LIN {X 0,Y 474.588,Z 296.363,A -85,B 0,C 180,E1 -7327.385,E2 -7327.385} C_VEL
LIN {X 0,Y 474.608,Z 296.362,A -85,B 0,C 180,E1 -7329.644,E2 -7329.644} C_VEL
LIN {X 0,Y 474.585,Z 296.364,A -85,B 0,C 180,E1 -7332.938,E2 -7332.938} C_VEL
LIN {X 0,Y 474.607,Z 296.362,A -85,B 0,C 180,E1 -7335.895,E2 -7335.895} C_VEL
LIN {X 0,Y 474.626,Z 296.36,A -85,B 0,C 180,E1 -7339.042,E2 -7339.042} C_VEL
LIN {X 0,Y 474.611,Z 296.36,A -85,B 0,C 180,E1 -7341.705,E2 -7341.705} C_VEL
LIN {X 0,Y 474.626,Z 296.367,A -85,B 0,C 180,E1 -7344.725,E2 -7344.725} C_VEL
LIN {X 0,Y 474.639,Z 296.356,A -85,B 0,C 180,E1 -7347.788,E2 -7347.788} C_VEL
LIN {X 0,Y 474.611,Z 296.367,A -85,B 0,C 180,E1 -7350.888,E2 -7350.888} C_VEL
LIN {X 0,Y 474.616,Z 296.361,A -85,B 0,C 180,E1 -7353.626,E2 -7353.626} C_VEL
LIN {X 0,Y 474.638,Z 296.358,A -85,B 0,C 180,E1 -7356.642,E2 -7356.642} C_VEL
LIN {X 0,Y 474.658,Z 296.354,A -85,B 0,C 180,E1 -7360.089,E2 -7360.089} C_VEL
LIN {X 0,Y 474.642,Z 296.357,A -85,B 0,C 180,E1 -7362.774,E2 -7362.774} C_VEL
LIN {X 0,Y 474.65,Z 296.362,A -85,B 0,C 180,E1 -7365.421,E2 -7365.421} C_VEL
LIN {X 0,Y 474.708,Z 296.351,A -85,B 0,C 180,E1 -7368.037,E2 -7368.037} C_VEL
LIN {X 0,Y 474.707,Z 296.352,A -85,B 0,C 180,E1 -7371.486,E2 -7371.486} C_VEL
LIN {X 0,Y 474.768,Z 296.347,A -85,B 0,C 180,E1 -7374.052,E2 -7374.052} C_VEL
LIN {X 0,Y 474.886,Z 296.327,A -85,B 0,C 180,E1 -7377.455,E2 -7377.455} C_VEL
LIN {X 0,Y 474.913,Z 296.33,A -85,B 0,C 180,E1 -7380,E2 -7380} C_VEL
LIN {X 0,Y 474.887,Z 296.329,A -85,B 0,C 180,E1 -7382.544,E2 -7382.544} C_VEL
LIN {X 0,Y 474.752,Z 296.346,A -85,B 0,C 180,E1 -7385.948,E2 -7385.948} C_VEL
LIN {X 0,Y 474.715,Z 296.355,A -85,B 0,C 180,E1 -7388.514,E2 -7388.514} C_VEL
LIN {X 0,Y 474.707,Z 296.349,A -85,B 0,C 180,E1 -7391.962,E2 -7391.962} C_VEL
LIN {X 0,Y 474.703,Z 296.349,A -85,B 0,C 180,E1 -7395.455,E2 -7395.455} C_VEL
LIN {X 0,Y 474.665,Z 296.359,A -85,B 0,C 180,E1 -7399.01,E2 -7399.01} C_VEL
LIN {X 0,Y 474.591,Z 296.363,A -85,B 0,C 180,E1 -7401.729,E2 -7401.729} C_VEL
LIN {X 0,Y 474.638,Z 296.358,A -85,B 0,C 180,E1 -7404.494,E2 -7404.494} C_VEL
LIN {X 0,Y 474.639,Z 296.363,A -85,B 0,C 180,E1 -7407.324,E2 -7407.324} C_VEL
LIN {X 0,Y 474.604,Z 296.361,A -85,B 0,C 180,E1 -7410.23,E2 -7410.23} C_VEL
LIN {X 0,Y 474.627,Z 296.364,A -85,B 0,C 180,E1 -7413.221,E2 -7413.221} C_VEL
LIN {X 0,Y 474.586,Z 296.363,A -85,B 0,C 180,E1 -7416.324,E2 -7416.324} C_VEL
LIN {X 0,Y 474.628,Z 296.366,A -85,B 0,C 180,E1 -7419.547,E2 -7419.547} C_VEL
LIN {X 0,Y 474.602,Z 296.363,A -85,B 0,C 180,E1 -7422.233,E2 -7422.233} C_VEL
LIN {X 0,Y 474.618,Z 296.361,A -85,B 0,C 180,E1 -7425.297,E2 -7425.297} C_VEL
LIN {X 0,Y 474.616,Z 296.364,A -85,B 0,C 180,E1 -7428.214,E2 -7428.214} C_VEL
LIN {X 0,Y 474.61,Z 296.362,A -85,B 0,C 180,E1 -7431.542,E2 -7431.542} C_VEL
LIN {X 0,Y 474.624,Z 296.36,A -85,B 0,C 180,E1 -7434.725,E2 -7434.725} C_VEL
LIN {X 0,Y 474.637,Z 296.358,A -85,B 0,C 180,E1 -7437.787,E2 -7437.787} C_VEL
LIN {X 0,Y 474.609,Z 296.363,A -85,B 0,C 180,E1 -7440.888,E2 -7440.888} C_VEL
LIN {X 0,Y 474.614,Z 296.359,A -85,B 0,C 180,E1 -7443.625,E2 -7443.625} C_VEL
LIN {X 0,Y 474.635,Z 296.366,A -85,B 0,C 180,E1 -7446.641,E2 -7446.641} C_VEL
LIN {X 0,Y 474.654,Z 296.355,A -85,B 0,C 180,E1 -7450.089,E2 -7450.089} C_VEL
LIN {X 0,Y 474.646,Z 296.356,A -85,B 0,C 180,E1 -7451.662,E2 -7451.662} C_VEL
LIN {X 0,Y 473.977,Z 296.442,A -85,B 0,C 180,E1 -7452.371,E2 -7452.371} C_VEL
LIN {X 0,Y 471.13,Z 296.799,A -85,B 0,C 180,E1 -7453.523,E2 -7453.523} C_VEL
LIN {X 0,Y 468.721,Z 297.102,A -85,B 0,C 180,E1 -7454.451,E2 -7454.451} C_VEL
LIN {X 0,Y 467.682,Z 297.229,A -85,B 0,C 180,E1 -7455.168,E2 -7455.168} C_VEL
LIN {X 0,Y 467.595,Z 297.237,A -85,B 0,C 180,E1 -7455.411,E2 -7455.411} C_VEL
LIN {X 0,Y 467.649,Z 297.23,A -85,B 0,C 180,E1 -7458.733,E2 -7458.733} C_VEL
LIN {X 0,Y 467.668,Z 297.234,A -85,B 0,C 180,E1 -7461.356,E2 -7461.356} C_VEL
LIN {X 0,Y 467.716,Z 297.278,A -85,B 0,C 180,E1 -7462.459,E2 -7462.459} C_VEL
LIN {X 0,Y 468.745,Z 303.411,A -85,B 0,C 180,E1 -7463.759,E2 -7463.759} C_VEL
LIN {X 0,Y 468.493,Z 316.288,A -85,B 0,C 180,E1 -7466.344,E2 -7466.344} C_VEL
LIN {X 0,Y 468.341,Z 320.083,A -85,B 0,C 180,E1 -7467.096,E2 -7467.096} C_VEL
LIN {X 0,Y 471.245,Z 335.027,A -85,B 0,C 180,E1 -7467.435,E2 -7467.435} C_VEL
LIN {X 0,Y 470.498,Z 427.693,A -85,B 0,C 180,E1 -7468.876,E2 -7468.876} C_VEL
LIN {X 0,Y 470.219,Z 440.684,A -85,B 0,C 180,E1 -7469.25,E2 -7469.25} C_VEL
LIN {X 0,Y 469.872,Z 453.221,A -85,B 0,C 180,E1 -7469.785,E2 -7469.785} C_VEL
LIN {X 0,Y 469.47,Z 464.404,A -85,B 0,C 180,E1 -7470.428,E2 -7470.428} C_VEL
LIN {X 0,Y 468.93,Z 475.979,A -85,B 0,C 180,E1 -7471.287,E2 -7471.287} C_VEL
LIN {X 0,Y 468.444,Z 486.385,A -85,B 0,C 180,E1 -7472.256,E2 -7472.256} C_VEL
LIN {X 0,Y 467.978,Z 494.922,A -85,B 0,C 180,E1 -7473.228,E2 -7473.228} C_VEL
LIN {X 0,Y 467.634,Z 502.784,A -85,B 0,C 180,E1 -7474.309,E2 -7474.309} C_VEL
LIN {X 0,Y 467.239,Z 510.504,A -85,B 0,C 180,E1 -7475.61,E2 -7475.61} C_VEL
LIN {X 0,Y 467.086,Z 516.68,A -85,B 0,C 180,E1 -7476.913,E2 -7476.913} C_VEL
LIN {X 0,Y 466.88,Z 521.614,A -85,B 0,C 180,E1 -7478.221,E2 -7478.221} C_VEL
LIN {X 0,Y 466.723,Z 525.428,A -85,B 0,C 180,E1 -7479.534,E2 -7479.534} C_VEL
LIN {X 0,Y 466.689,Z 527.392,A -85,B 0,C 180,E1 -7480.41,E2 -7480.41} C_VEL
LIN {X 0,Y 466.645,Z 529.579,A -85,B 0,C 180,E1 -7481.779,E2 -7481.779} C_VEL
LIN {X 0,Y 466.555,Z 530.699,A -85,B 0,C 180,E1 -7483.058,E2 -7483.058} C_VEL
LIN {X 0,Y 466.525,Z 530.982,A -85,B 0,C 180,E1 -7483.947,E2 -7483.947} C_VEL
LIN {X 0,Y 466.613,Z 530.508,A -85,B 0,C 180,E1 -7485.432,E2 -7485.432} C_VEL
LIN {X 0,Y 466.545,Z 529.246,A -85,B 0,C 180,E1 -7486.631,E2 -7486.631} C_VEL
LIN {X 0,Y 466.636,Z 527.819,A -85,B 0,C 180,E1 -7487.53,E2 -7487.53} C_VEL
LIN {X 0,Y 466.785,Z 524.885,A -85,B 0,C 180,E1 -7488.841,E2 -7488.841} C_VEL
LIN {X 0,Y 466.937,Z 520.549,A -85,B 0,C 180,E1 -7490.253,E2 -7490.253} C_VEL
LIN {X 0,Y 467.135,Z 515.016,A -85,B 0,C 180,E1 -7491.628,E2 -7491.628} C_VEL
LIN {X 0,Y 467.489,Z 507.978,A -85,B 0,C 180,E1 -7493.008,E2 -7493.008} C_VEL
LIN {X 0,Y 467.83,Z 500.694,A -85,B 0,C 180,E1 -7494.164,E2 -7494.164} C_VEL
LIN {X 0,Y 468.293,Z 491.797,A -85,B 0,C 180,E1 -7495.322,E2 -7495.322} C_VEL
LIN {X 0,Y 468.754,Z 482.224,A -85,B 0,C 180,E1 -7496.333,E2 -7496.333} C_VEL
LIN {X 0,Y 469.341,Z 470.875,A -85,B 0,C 180,E1 -7497.295,E2 -7497.295} C_VEL
LIN {X 0,Y 469.835,Z 459.618,A -85,B 0,C 180,E1 -7498.049,E2 -7498.049} C_VEL
LIN {X 0,Y 470.194,Z 448.276,A -85,B 0,C 180,E1 -7498.635,E2 -7498.635} C_VEL
LIN {X 0,Y 470.537,Z 434.709,A -85,B 0,C 180,E1 -7499.131,E2 -7499.131} C_VEL
LIN {X 0,Y 470.768,Z 421.895,A -85,B 0,C 180,E1 -7499.422,E2 -7499.422} C_VEL
LIN {X 0,Y 471.51,Z 335.217,A -85,B 0,C 180,E1 -7500.76,E2 -7500.76} C_VEL
LIN {X 0,Y 468.488,Z 319.878,A -85,B 0,C 180,E1 -7501.148,E2 -7501.148} C_VEL
LIN {X 0,Y 468.923,Z 305.629,A -85,B 0,C 180,E1 -7503.915,E2 -7503.915} C_VEL
LIN {X 0,Y 468.16,Z 300.097,A -85,B 0,C 180,E1 -7505.043,E2 -7505.043} C_VEL
LIN {X 0,Y 467.563,Z 297.245,A -85,B 0,C 180,E1 -7505.664,E2 -7505.664} C_VEL
LIN {X 0,Y 467.546,Z 297.246,A -85,B 0,C 180,E1 -7509.147,E2 -7509.147} C_VEL
LIN {X 0,Y 467.56,Z 297.242,A -85,B 0,C 180,E1 -7511.403,E2 -7511.403} C_VEL
LIN {X 0,Y 467.558,Z 297.247,A -85,B 0,C 180,E1 -7514.947,E2 -7514.947} C_VEL
LIN {X 0,Y 467.535,Z 297.244,A -85,B 0,C 180,E1 -7517.438,E2 -7517.438} C_VEL
LIN {X 0,Y 467.555,Z 297.241,A -85,B 0,C 180,E1 -7520.048,E2 -7520.048} C_VEL
LIN {X 0,Y 467.52,Z 297.248,A -85,B 0,C 180,E1 -7523.037,E2 -7523.037} C_VEL
LIN {X 0,Y 467.558,Z 297.23,A -85,B 0,C 180,E1 -7526.21,E2 -7526.21} C_VEL
LIN {X 0,Y 467.559,Z 297.245,A -85,B 0,C 180,E1 -7529.266,E2 -7529.266} C_VEL
LIN {X 0,Y 467.594,Z 297.236,A -85,B 0,C 180,E1 -7532.469,E2 -7532.469} C_VEL
LIN {X 0,Y 467.545,Z 297.241,A -85,B 0,C 180,E1 -7535.11,E2 -7535.11} C_VEL
LIN {X 0,Y 467.524,Z 297.247,A -85,B 0,C 180,E1 -7537.926,E2 -7537.926} C_VEL
LIN {X 0,Y 467.61,Z 297.232,A -85,B 0,C 180,E1 -7540.692,E2 -7540.692} C_VEL
LIN {X 0,Y 467.595,Z 297.238,A -85,B 0,C 180,E1 -7544.304,E2 -7544.304} C_VEL
LIN {X 0,Y 467.638,Z 297.23,A -85,B 0,C 180,E1 -7547.854,E2 -7547.854} C_VEL
LIN {X 0,Y 467.619,Z 297.227,A -85,B 0,C 180,E1 -7551.356,E2 -7551.356} C_VEL
LIN {X 0,Y 467.681,Z 297.227,A -85,B 0,C 180,E1 -7553.962,E2 -7553.962} C_VEL
LIN {X 0,Y 467.778,Z 297.207,A -85,B 0,C 180,E1 -7557.417,E2 -7557.417} C_VEL
LIN {X 0,Y 467.835,Z 297.208,A -85,B 0,C 180,E1 -7560,E2 -7560} C_VEL
LIN {X 0,Y 467.799,Z 297.21,A -85,B 0,C 180,E1 -7562.583,E2 -7562.583} C_VEL
LIN {X 0,Y 467.711,Z 297.221,A -85,B 0,C 180,E1 -7566.038,E2 -7566.038} C_VEL
LIN {X 0,Y 467.644,Z 297.229,A -85,B 0,C 180,E1 -7568.644,E2 -7568.644} C_VEL
LIN {X 0,Y 467.647,Z 297.227,A -85,B 0,C 180,E1 -7572.146,E2 -7572.146} C_VEL
LIN {X 0,Y 467.64,Z 297.228,A -85,B 0,C 180,E1 -7575.885,E2 -7575.885} C_VEL
LIN {X 0,Y 467.612,Z 297.236,A -85,B 0,C 180,E1 -7579.308,E2 -7579.308} C_VEL
LIN {X 0,Y 467.522,Z 297.241,A -85,B 0,C 180,E1 -7582.075,E2 -7582.075} C_VEL
LIN {X 0,Y 467.552,Z 297.242,A -85,B 0,C 180,E1 -7584.891,E2 -7584.891} C_VEL
LIN {X 0,Y 467.571,Z 297.238,A -85,B 0,C 180,E1 -7587.772,E2 -7587.772} C_VEL
LIN {X 0,Y 467.56,Z 297.243,A -85,B 0,C 180,E1 -7591.045,E2 -7591.045} C_VEL
LIN {X 0,Y 467.581,Z 297.237,A -85,B 0,C 180,E1 -7594.243,E2 -7594.243} C_VEL
LIN {X 0,Y 467.536,Z 297.245,A -85,B 0,C 180,E1 -7597.186,E2 -7597.186} C_VEL
LIN {X 0,Y 467.553,Z 297.243,A -85,B 0,C 180,E1 -7600.267,E2 -7600.267} C_VEL
LIN {X 0,Y 467.555,Z 297.234,A -85,B 0,C 180,E1 -7602.564,E2 -7602.564} C_VEL
LIN {X 0,Y 467.56,Z 297.239,A -85,B 0,C 180,E1 -7605.053,E2 -7605.053} C_VEL
LIN {X 0,Y 467.569,Z 297.242,A -85,B 0,C 180,E1 -7608.598,E2 -7608.598} C_VEL
LIN {X 0,Y 467.559,Z 297.247,A -85,B 0,C 180,E1 -7611.956,E2 -7611.956} C_VEL
LIN {X 0,Y 467.559,Z 297.238,A -85,B 0,C 180,E1 -7615.168,E2 -7615.168} C_VEL
LIN {X 0,Y 467.58,Z 297.242,A -85,B 0,C 180,E1 -7618.261,E2 -7618.261} C_VEL
LIN {X 0,Y 467.571,Z 297.241,A -85,B 0,C 180,E1 -7621.251,E2 -7621.251} C_VEL
LIN {X 0,Y 467.6,Z 297.247,A -85,B 0,C 180,E1 -7624.263,E2 -7624.263} C_VEL
LIN {X 0,Y 469.688,Z 308.038,A -85,B 0,C 180,E1 -7626.406,E2 -7626.406} C_VEL
LIN {X 0,Y 469.625,Z 314.378,A -85,B 0,C 180,E1 -7627.568,E2 -7627.568} C_VEL
LIN {X 0,Y 468.868,Z 332.121,A -85,B 0,C 180,E1 -7630.747,E2 -7630.747} C_VEL
LIN {X 0,Y 468.377,Z 344.572,A -85,B 0,C 180,E1 -7632.917,E2 -7632.917} C_VEL
LIN {X 0,Y 471.377,Z 363.661,A -85,B 0,C 180,E1 -7633.339,E2 -7633.339} C_VEL
LIN {X 0,Y 470.684,Z 453.085,A -85,B 0,C 180,E1 -7634.743,E2 -7634.743} C_VEL
LIN {X 0,Y 470.28,Z 465.397,A -85,B 0,C 180,E1 -7635.09,E2 -7635.09} C_VEL
LIN {X 0,Y 469.805,Z 478.772,A -85,B 0,C 180,E1 -7635.656,E2 -7635.656} C_VEL
LIN {X 0,Y 469.326,Z 490.801,A -85,B 0,C 180,E1 -7636.359,E2 -7636.359} C_VEL
LIN {X 0,Y 468.741,Z 502.11,A -85,B 0,C 180,E1 -7637.209,E2 -7637.209} C_VEL
LIN {X 0,Y 468.242,Z 512.66,A -85,B 0,C 180,E1 -7638.201,E2 -7638.201} C_VEL
LIN {X 0,Y 467.83,Z 521.149,A -85,B 0,C 180,E1 -7639.178,E2 -7639.178} C_VEL
LIN {X 0,Y 467.383,Z 530.356,A -85,B 0,C 180,E1 -7640.48,E2 -7640.48} C_VEL
LIN {X 0,Y 467.066,Z 537.769,A -85,B 0,C 180,E1 -7641.782,E2 -7641.782} C_VEL
LIN {X 0,Y 466.859,Z 543.725,A -85,B 0,C 180,E1 -7643.084,E2 -7643.084} C_VEL
LIN {X 0,Y 466.761,Z 548.434,A -85,B 0,C 180,E1 -7644.384,E2 -7644.384} C_VEL
LIN {X 0,Y 466.646,Z 552.03,A -85,B 0,C 180,E1 -7645.682,E2 -7645.682} C_VEL
LIN {X 0,Y 466.688,Z 553.885,A -85,B 0,C 180,E1 -7646.547,E2 -7646.547} C_VEL
LIN {X 0,Y 466.662,Z 555.276,A -85,B 0,C 180,E1 -7647.411,E2 -7647.411} C_VEL
LIN {X 0,Y 466.618,Z 556.874,A -85,B 0,C 180,E1 -7649.138,E2 -7649.138} C_VEL
LIN {X 0,Y 466.599,Z 557.083,A -85,B 0,C 180,E1 -7650.001,E2 -7650.001} C_VEL
LIN {X 0,Y 466.618,Z 556.861,A -85,B 0,C 180,E1 -7650.864,E2 -7650.864} C_VEL
LIN {X 0,Y 466.662,Z 555.249,A -85,B 0,C 180,E1 -7652.59,E2 -7652.59} C_VEL
LIN {X 0,Y 466.689,Z 553.842,A -85,B 0,C 180,E1 -7653.454,E2 -7653.454} C_VEL
LIN {X 0,Y 466.689,Z 550.89,A -85,B 0,C 180,E1 -7654.752,E2 -7654.752} C_VEL
LIN {X 0,Y 466.753,Z 546.891,A -85,B 0,C 180,E1 -7656.051,E2 -7656.051} C_VEL
LIN {X 0,Y 466.944,Z 540.735,A -85,B 0,C 180,E1 -7657.568,E2 -7657.568} C_VEL
LIN {X 0,Y 467.196,Z 534.013,A -85,B 0,C 180,E1 -7658.871,E2 -7658.871} C_VEL
LIN {X 0,Y 467.569,Z 525.67,A -85,B 0,C 180,E1 -7660.173,E2 -7660.173} C_VEL
LIN {X 0,Y 467.985,Z 517.088,A -85,B 0,C 180,E1 -7661.259,E2 -7661.259} C_VEL
LIN {X 0,Y 468.513,Z 506.921,A -85,B 0,C 180,E1 -7662.304,E2 -7662.304} C_VEL
LIN {X 0,Y 468.92,Z 495.985,A -85,B 0,C 180,E1 -7663.213,E2 -7663.213} C_VEL
LIN {X 0,Y 469.446,Z 484.41,A -85,B 0,C 180,E1 -7663.97,E2 -7663.97} C_VEL
LIN {X 0,Y 469.922,Z 472.385,A -85,B 0,C 180,E1 -7664.564,E2 -7664.564} C_VEL
LIN {X 0,Y 470.307,Z 460.279,A -85,B 0,C 180,E1 -7664.994,E2 -7664.994} C_VEL
LIN {X 0,Y 470.559,Z 447.109,A -85,B 0,C 180,E1 -7665.291,E2 -7665.291} C_VEL
LIN {X 0,Y 471.018,Z 362.015,A -85,B 0,C 180,E1 -7666.599,E2 -7666.599} C_VEL
LIN {X 0,Y 468.314,Z 344.575,A -85,B 0,C 180,E1 -7666.966,E2 -7666.966} C_VEL
LIN {X 0,Y 468.937,Z 327.705,A -85,B 0,C 180,E1 -7669.936,E2 -7669.936} C_VEL
LIN {X 0,Y 469.61,Z 312.347,A -85,B 0,C 180,E1 -7672.667,E2 -7672.667} C_VEL
LIN {X 0,Y 469.523,Z 307.199,A -85,B 0,C 180,E1 -7673.604,E2 -7673.604} C_VEL
LIN {X 0,Y 467.608,Z 297.241,A -85,B 0,C 180,E1 -7675.557,E2 -7675.557} C_VEL
LIN {X 0,Y 467.62,Z 297.239,A -85,B 0,C 180,E1 -7677.77,E2 -7677.77} C_VEL
LIN {X 0,Y 467.571,Z 297.237,A -85,B 0,C 180,E1 -7681.045,E2 -7681.045} C_VEL
LIN {X 0,Y 467.592,Z 297.239,A -85,B 0,C 180,E1 -7684.242,E2 -7684.242} C_VEL
LIN {X 0,Y 467.546,Z 297.24,A -85,B 0,C 180,E1 -7687.186,E2 -7687.186} C_VEL
LIN {X 0,Y 467.563,Z 297.246,A -85,B 0,C 180,E1 -7690.267,E2 -7690.267} C_VEL
LIN {X 0,Y 467.564,Z 297.243,A -85,B 0,C 180,E1 -7692.564,E2 -7692.564} C_VEL
LIN {X 0,Y 467.569,Z 297.238,A -85,B 0,C 180,E1 -7695.053,E2 -7695.053} C_VEL
LIN {X 0,Y 467.577,Z 297.244,A -85,B 0,C 180,E1 -7698.597,E2 -7698.597} C_VEL
LIN {X 0,Y 467.566,Z 297.238,A -85,B 0,C 180,E1 -7701.955,E2 -7701.955} C_VEL
LIN {X 0,Y 467.566,Z 297.241,A -85,B 0,C 180,E1 -7705.167,E2 -7705.167} C_VEL
LIN {X 0,Y 467.586,Z 297.236,A -85,B 0,C 180,E1 -7708.26,E2 -7708.26} C_VEL
LIN {X 0,Y 467.56,Z 297.243,A -85,B 0,C 180,E1 -7711.249,E2 -7711.249} C_VEL
LIN {X 0,Y 467.586,Z 297.235,A -85,B 0,C 180,E1 -7714.158,E2 -7714.158} C_VEL
LIN {X 0,Y 467.579,Z 297.241,A -85,B 0,C 180,E1 -7716.996,E2 -7716.996} C_VEL
LIN {X 0,Y 467.626,Z 297.233,A -85,B 0,C 180,E1 -7719.777,E2 -7719.777} C_VEL
LIN {X 0,Y 467.602,Z 297.233,A -85,B 0,C 180,E1 -7722.506,E2 -7722.506} C_VEL
LIN {X 0,Y 467.608,Z 297.236,A -85,B 0,C 180,E1 -7725.196,E2 -7725.196} C_VEL
LIN {X 0,Y 467.66,Z 297.232,A -85,B 0,C 180,E1 -7727.854,E2 -7727.854} C_VEL
LIN {X 0,Y 467.666,Z 297.228,A -85,B 0,C 180,E1 -7731.357,E2 -7731.357} C_VEL
LIN {X 0,Y 467.732,Z 297.225,A -85,B 0,C 180,E1 -7733.962,E2 -7733.962} C_VEL
LIN {X 0,Y 467.851,Z 297.203,A -85,B 0,C 180,E1 -7737.417,E2 -7737.417} C_VEL
LIN {X 0,Y 467.883,Z 297.205,A -85,B 0,C 180,E1 -7740,E2 -7740} C_VEL
LIN {X 0,Y 467.853,Z 297.205,A -85,B 0,C 180,E1 -7742.583,E2 -7742.583} C_VEL
LIN {X 0,Y 467.715,Z 297.223,A -85,B 0,C 180,E1 -7746.038,E2 -7746.038} C_VEL
LIN {X 0,Y 467.673,Z 297.23,A -85,B 0,C 180,E1 -7748.643,E2 -7748.643} C_VEL
LIN {X 0,Y 467.659,Z 297.229,A -85,B 0,C 180,E1 -7752.145,E2 -7752.145} C_VEL
LIN {X 0,Y 467.642,Z 297.228,A -85,B 0,C 180,E1 -7755.695,E2 -7755.695} C_VEL
LIN {X 0,Y 467.625,Z 297.233,A -85,B 0,C 180,E1 -7759.307,E2 -7759.307} C_VEL
LIN {X 0,Y 467.537,Z 297.241,A -85,B 0,C 180,E1 -7762.074,E2 -7762.074} C_VEL
LIN {X 0,Y 467.586,Z 297.241,A -85,B 0,C 180,E1 -7764.888,E2 -7764.888} C_VEL
LIN {X 0,Y 467.582,Z 297.237,A -85,B 0,C 180,E1 -7767.771,E2 -7767.771} C_VEL
LIN {X 0,Y 467.569,Z 297.242,A -85,B 0,C 180,E1 -7771.044,E2 -7771.044} C_VEL
LIN {X 0,Y 467.579,Z 297.236,A -85,B 0,C 180,E1 -7774.24,E2 -7774.24} C_VEL
LIN {X 0,Y 467.545,Z 297.244,A -85,B 0,C 180,E1 -7777.185,E2 -7777.185} C_VEL
LIN {X 0,Y 467.572,Z 297.238,A -85,B 0,C 180,E1 -7780.265,E2 -7780.265} C_VEL
LIN {X 0,Y 467.55,Z 297.248,A -85,B 0,C 180,E1 -7783.745,E2 -7783.745} C_VEL
LIN {X 0,Y 467.55,Z 297.243,A -85,B 0,C 180,E1 -7786.254,E2 -7786.254} C_VEL
LIN {X 0,Y 467.576,Z 297.237,A -85,B 0,C 180,E1 -7788.723,E2 -7788.723} C_VEL
LIN {X 0,Y 467.563,Z 297.245,A -85,B 0,C 180,E1 -7791.955,E2 -7791.955} C_VEL
LIN {X 0,Y 467.564,Z 297.238,A -85,B 0,C 180,E1 -7795.167,E2 -7795.167} C_VEL
LIN {X 0,Y 467.585,Z 297.243,A -85,B 0,C 180,E1 -7798.259,E2 -7798.259} C_VEL
LIN {X 0,Y 467.557,Z 297.239,A -85,B 0,C 180,E1 -7801.248,E2 -7801.248} C_VEL
LIN {X 0,Y 467.584,Z 297.238,A -85,B 0,C 180,E1 -7804.158,E2 -7804.158} C_VEL
LIN {X 0,Y 467.577,Z 297.24,A -85,B 0,C 180,E1 -7806.995,E2 -7806.995} C_VEL
LIN {X 0,Y 467.622,Z 297.23,A -85,B 0,C 180,E1 -7809.777,E2 -7809.777} C_VEL
LIN {X 0,Y 467.596,Z 297.237,A -85,B 0,C 180,E1 -7812.506,E2 -7812.506} C_VEL
LIN {X 0,Y 467.604,Z 297.239,A -85,B 0,C 180,E1 -7815.196,E2 -7815.196} C_VEL
LIN {X 0,Y 467.595,Z 297.237,A -85,B 0,C 180,E1 -7815.411,E2 -7815.411} C_VEL
LIN {X 0,Y 466.923,Z 297.318,A -85,B 0,C 180,E1 -7816.13,E2 -7816.13} C_VEL
LIN {X 0,Y 464.081,Z 297.677,A -85,B 0,C 180,E1 -7817.299,E2 -7817.299} C_VEL
LIN {X 0,Y 461.682,Z 297.973,A -85,B 0,C 180,E1 -7818.241,E2 -7818.241} C_VEL
LIN {X 0,Y 460.654,Z 298.105,A -85,B 0,C 180,E1 -7818.969,E2 -7818.969} C_VEL
LIN {X 0,Y 460.571,Z 298.112,A -85,B 0,C 180,E1 -7819.215,E2 -7819.215} C_VEL
LIN {X 0,Y 460.665,Z 298.117,A -85,B 0,C 180,E1 -7822.298,E2 -7822.298} C_VEL
LIN {X 0,Y 461.744,Z 304.496,A -85,B 0,C 180,E1 -7823.664,E2 -7823.664} C_VEL
LIN {X 0,Y 461.503,Z 317.416,A -85,B 0,C 180,E1 -7826.288,E2 -7826.288} C_VEL
LIN {X 0,Y 461.362,Z 320.278,A -85,B 0,C 180,E1 -7826.861,E2 -7826.861} C_VEL
LIN {X 0,Y 464.396,Z 335.7,A -85,B 0,C 180,E1 -7827.213,E2 -7827.213} C_VEL
LIN {X 0,Y 463.617,Z 427.932,A -85,B 0,C 180,E1 -7828.669,E2 -7828.669} C_VEL
LIN {X 0,Y 463.324,Z 440.909,A -85,B 0,C 180,E1 -7829.049,E2 -7829.049} C_VEL
LIN {X 0,Y 462.947,Z 453.983,A -85,B 0,C 180,E1 -7829.619,E2 -7829.619} C_VEL
LIN {X 0,Y 462.468,Z 465.814,A -85,B 0,C 180,E1 -7830.326,E2 -7830.326} C_VEL
LIN {X 0,Y 461.928,Z 477.17,A -85,B 0,C 180,E1 -7831.198,E2 -7831.198} C_VEL
LIN {X 0,Y 461.422,Z 487.417,A -85,B 0,C 180,E1 -7832.181,E2 -7832.181} C_VEL
LIN {X 0,Y 460.902,Z 496.647,A -85,B 0,C 180,E1 -7833.277,E2 -7833.277} C_VEL
LIN {X 0,Y 460.497,Z 505.593,A -85,B 0,C 180,E1 -7834.595,E2 -7834.595} C_VEL
LIN {X 0,Y 460.153,Z 512.823,A -85,B 0,C 180,E1 -7835.917,E2 -7835.917} C_VEL
LIN {X 0,Y 460,Z 517.706,A -85,B 0,C 180,E1 -7837.02,E2 -7837.02} C_VEL
LIN {X 0,Y 459.77,Z 522.47,A -85,B 0,C 180,E1 -7838.349,E2 -7838.349} C_VEL
LIN {X 0,Y 459.618,Z 526.12,A -85,B 0,C 180,E1 -7839.682,E2 -7839.682} C_VEL
LIN {X 0,Y 459.609,Z 527.998,A -85,B 0,C 180,E1 -7840.573,E2 -7840.573} C_VEL
LIN {X 0,Y 459.565,Z 529.879,A -85,B 0,C 180,E1 -7841.838,E2 -7841.838} C_VEL
LIN {X 0,Y 459.443,Z 531.012,A -85,B 0,C 180,E1 -7843.264,E2 -7843.264} C_VEL
LIN {X 0,Y 459.449,Z 531.188,A -85,B 0,C 180,E1 -7844.166,E2 -7844.166} C_VEL
LIN {X 0,Y 459.517,Z 530.669,A -85,B 0,C 180,E1 -7845.52,E2 -7845.52} C_VEL
LIN {X 0,Y 459.476,Z 529.173,A -85,B 0,C 180,E1 -7846.894,E2 -7846.894} C_VEL
LIN {X 0,Y 459.703,Z 525.916,A -85,B 0,C 180,E1 -7848.583,E2 -7848.583} C_VEL
LIN {X 0,Y 459.832,Z 521.589,A -85,B 0,C 180,E1 -7850.113,E2 -7850.113} C_VEL
LIN {X 0,Y 460.066,Z 516.344,A -85,B 0,C 180,E1 -7851.507,E2 -7851.507} C_VEL
LIN {X 0,Y 460.413,Z 509.605,A -85,B 0,C 180,E1 -7852.907,E2 -7852.907} C_VEL
LIN {X 0,Y 460.842,Z 501.06,A -85,B 0,C 180,E1 -7854.314,E2 -7854.314} C_VEL
LIN {X 0,Y 461.343,Z 492.333,A -85,B 0,C 180,E1 -7855.474,E2 -7855.474} C_VEL
LIN {X 0,Y 461.844,Z 482.324,A -85,B 0,C 180,E1 -7856.551,E2 -7856.551} C_VEL
LIN {X 0,Y 462.463,Z 471.417,A -85,B 0,C 180,E1 -7857.49,E2 -7857.49} C_VEL
LIN {X 0,Y 463.019,Z 459.269,A -85,B 0,C 180,E1 -7858.314,E2 -7858.314} C_VEL
LIN {X 0,Y 463.432,Z 447.401,A -85,B 0,C 180,E1 -7858.92,E2 -7858.92} C_VEL
LIN {X 0,Y 463.74,Z 434.811,A -85,B 0,C 180,E1 -7859.382,E2 -7859.382} C_VEL
LIN {X 0,Y 463.979,Z 421.929,A -85,B 0,C 180,E1 -7859.677,E2 -7859.677} C_VEL
LIN {X 0,Y 464.718,Z 335.728,A -85,B 0,C 180,E1 -7861.03,E2 -7861.03} C_VEL
LIN {X 0,Y 461.576,Z 320.073,A -85,B 0,C 180,E1 -7861.439,E2 -7861.439} C_VEL
LIN {X 0,Y 462.01,Z 307.102,A -85,B 0,C 180,E1 -7863.988,E2 -7863.988} C_VEL
LIN {X 0,Y 461.375,Z 302.265,A -85,B 0,C 180,E1 -7864.987,E2 -7864.987} C_VEL
LIN {X 0,Y 460.498,Z 298.125,A -85,B 0,C 180,E1 -7865.905,E2 -7865.905} C_VEL
LIN {X 0,Y 460.498,Z 298.126,A -85,B 0,C 180,E1 -7868.891,E2 -7868.891} C_VEL
LIN {X 0,Y 460.506,Z 298.12,A -85,B 0,C 180,E1 -7871.599,E2 -7871.599} C_VEL
LIN {X 0,Y 460.504,Z 298.123,A -85,B 0,C 180,E1 -7874.589,E2 -7874.589} C_VEL
LIN {X 0,Y 460.482,Z 298.122,A -85,B 0,C 180,E1 -7877.814,E2 -7877.814} C_VEL
LIN {X 0,Y 460.521,Z 298.123,A -85,B 0,C 180,E1 -7881.104,E2 -7881.104} C_VEL
LIN {X 0,Y 460.5,Z 298.12,A -85,B 0,C 180,E1 -7884.554,E2 -7884.554} C_VEL
LIN {X 0,Y 460.516,Z 298.121,A -85,B 0,C 180,E1 -7887.715,E2 -7887.715} C_VEL
LIN {X 0,Y 460.516,Z 298.115,A -85,B 0,C 180,E1 -7890.768,E2 -7890.768} C_VEL
LIN {X 0,Y 460.505,Z 298.121,A -85,B 0,C 180,E1 -7893.731,E2 -7893.731} C_VEL
LIN {X 0,Y 460.534,Z 298.114,A -85,B 0,C 180,E1 -7896.624,E2 -7896.624} C_VEL
LIN {X 0,Y 460.54,Z 298.116,A -85,B 0,C 180,E1 -7899.452,E2 -7899.452} C_VEL
LIN {X 0,Y 460.515,Z 298.119,A -85,B 0,C 180,E1 -7902.229,E2 -7902.229} C_VEL
LIN {X 0,Y 460.532,Z 298.114,A -85,B 0,C 180,E1 -7904.964,E2 -7904.964} C_VEL
LIN {X 0,Y 460.593,Z 298.105,A -85,B 0,C 180,E1 -7907.666,E2 -7907.666} C_VEL
LIN {X 0,Y 460.574,Z 298.104,A -85,B 0,C 180,E1 -7911.223,E2 -7911.223} C_VEL
LIN {X 0,Y 460.648,Z 298.102,A -85,B 0,C 180,E1 -7913.869,E2 -7913.869} C_VEL
LIN {X 0,Y 460.725,Z 298.086,A -85,B 0,C 180,E1 -7917.377,E2 -7917.377} C_VEL
LIN {X 0,Y 460.784,Z 298.086,A -85,B 0,C 180,E1 -7920,E2 -7920} C_VEL
LIN {X 0,Y 460.743,Z 298.089,A -85,B 0,C 180,E1 -7922.623,E2 -7922.623} C_VEL
LIN {X 0,Y 460.677,Z 298.098,A -85,B 0,C 180,E1 -7926.131,E2 -7926.131} C_VEL
LIN {X 0,Y 460.594,Z 298.108,A -85,B 0,C 180,E1 -7928.777,E2 -7928.777} C_VEL
LIN {X 0,Y 460.588,Z 298.108,A -85,B 0,C 180,E1 -7932.435,E2 -7932.435} C_VEL
LIN {X 0,Y 460.592,Z 298.105,A -85,B 0,C 180,E1 -7935.998,E2 -7935.998} C_VEL
LIN {X 0,Y 460.559,Z 298.111,A -85,B 0,C 180,E1 -7939.616,E2 -7939.616} C_VEL
LIN {X 0,Y 460.499,Z 298.116,A -85,B 0,C 180,E1 -7942.43,E2 -7942.43} C_VEL
LIN {X 0,Y 460.527,Z 298.116,A -85,B 0,C 180,E1 -7945.794,E2 -7945.794} C_VEL
LIN {X 0,Y 460.518,Z 298.114,A -85,B 0,C 180,E1 -7948.236,E2 -7948.236} C_VEL
LIN {X 0,Y 460.513,Z 298.121,A -85,B 0,C 180,E1 -7951.283,E2 -7951.283} C_VEL
LIN {X 0,Y 460.524,Z 298.115,A -85,B 0,C 180,E1 -7954.506,E2 -7954.506} C_VEL
LIN {X 0,Y 460.492,Z 298.126,A -85,B 0,C 180,E1 -7957.624,E2 -7957.624} C_VEL
LIN {X 0,Y 460.514,Z 298.119,A -85,B 0,C 180,E1 -7961.013,E2 -7961.013} C_VEL
LIN {X 0,Y 460.5,Z 298.119,A -85,B 0,C 180,E1 -7964.17,E2 -7964.17} C_VEL
LIN {X 0,Y 460.487,Z 298.123,A -85,B 0,C 180,E1 -7967.104,E2 -7967.104} C_VEL
LIN {X 0,Y 460.515,Z 298.126,A -85,B 0,C 180,E1 -7970.137,E2 -7970.137} C_VEL
LIN {X 0,Y 460.469,Z 298.125,A -85,B 0,C 180,E1 -7973.471,E2 -7973.471} C_VEL
LIN {X 0,Y 460.527,Z 298.12,A -85,B 0,C 180,E1 -7976.676,E2 -7976.676} C_VEL
LIN {X 0,Y 460.508,Z 298.124,A -85,B 0,C 180,E1 -7979.761,E2 -7979.761} C_VEL
LIN {X 0,Y 460.556,Z 298.119,A -85,B 0,C 180,E1 -7982.756,E2 -7982.756} C_VEL
LIN {X 0,Y 460.573,Z 298.26,A -85,B 0,C 180,E1 -7984.051,E2 -7984.051} C_VEL
LIN {X 0,Y 462.756,Z 309.272,A -85,B 0,C 180,E1 -7986.269,E2 -7986.269} C_VEL
LIN {X 0,Y 462.837,Z 314.333,A -85,B 0,C 180,E1 -7987.22,E2 -7987.22} C_VEL
LIN {X 0,Y 461.9,Z 333.056,A -85,B 0,C 180,E1 -7990.624,E2 -7990.624} C_VEL
LIN {X 0,Y 461.424,Z 344.098,A -85,B 0,C 180,E1 -7992.608,E2 -7992.608} C_VEL
LIN {X 0,Y 464.588,Z 363.787,A -85,B 0,C 180,E1 -7993.071,E2 -7993.071} C_VEL
LIN {X 0,Y 463.903,Z 452.611,A -85,B 0,C 180,E1 -7994.486,E2 -7994.486} C_VEL
LIN {X 0,Y 463.467,Z 465.012,A -85,B 0,C 180,E1 -7994.837,E2 -7994.837} C_VEL
LIN {X 0,Y 463.006,Z 477.87,A -85,B 0,C 180,E1 -7995.384,E2 -7995.384} C_VEL
LIN {X 0,Y 462.486,Z 489.293,A -85,B 0,C 180,E1 -7996.041,E2 -7996.041} C_VEL
LIN {X 0,Y 461.844,Z 501.253,A -85,B 0,C 180,E1 -7996.937,E2 -7996.937} C_VEL
LIN {X 0,Y 461.35,Z 511.572,A -85,B 0,C 180,E1 -7997.91,E2 -7997.91} C_VEL
LIN {X 0,Y 460.819,Z 521.086,A -85,B 0,C 180,E1 -7999.011,E2 -7999.011} C_VEL
LIN {X 0,Y 460.366,Z 530.25,A -85,B 0,C 180,E1 -8000.334,E2 -8000.334} C_VEL
LIN {X 0,Y 460.003,Z 537.638,A -85,B 0,C 180,E1 -8001.655,E2 -8001.655} C_VEL
LIN {X 0,Y 459.778,Z 543.577,A -85,B 0,C 180,E1 -8002.977,E2 -8002.977} C_VEL
LIN {X 0,Y 459.66,Z 548.275,A -85,B 0,C 180,E1 -8004.297,E2 -8004.297} C_VEL
LIN {X 0,Y 459.564,Z 551.862,A -85,B 0,C 180,E1 -8005.615,E2 -8005.615} C_VEL
LIN {X 0,Y 459.583,Z 553.709,A -85,B 0,C 180,E1 -8006.494,E2 -8006.494} C_VEL
LIN {X 0,Y 459.584,Z 555.093,A -85,B 0,C 180,E1 -8007.371,E2 -8007.371} C_VEL
LIN {X 0,Y 459.521,Z 556.682,A -85,B 0,C 180,E1 -8009.124,E2 -8009.124} C_VEL
LIN {X 0,Y 459.53,Z 556.884,A -85,B 0,C 180,E1 -8010.001,E2 -8010.001} C_VEL
LIN {X 0,Y 459.52,Z 556.038,A -85,B 0,C 180,E1 -8011.754,E2 -8011.754} C_VEL
LIN {X 0,Y 459.584,Z 555.034,A -85,B 0,C 180,E1 -8012.63,E2 -8012.63} C_VEL
LIN {X 0,Y 459.584,Z 553.617,A -85,B 0,C 180,E1 -8013.508,E2 -8013.508} C_VEL
LIN {X 0,Y 459.617,Z 550.656,A -85,B 0,C 180,E1 -8014.825,E2 -8014.825} C_VEL
LIN {X 0,Y 459.715,Z 545.599,A -85,B 0,C 180,E1 -8016.432,E2 -8016.432} C_VEL
LIN {X 0,Y 459.894,Z 539.456,A -85,B 0,C 180,E1 -8017.906,E2 -8017.906} C_VEL
LIN {X 0,Y 460.22,Z 532.49,A -85,B 0,C 180,E1 -8019.228,E2 -8019.228} C_VEL
LIN {X 0,Y 460.59,Z 523.746,A -85,B 0,C 180,E1 -8020.551,E2 -8020.551} C_VEL
LIN {X 0,Y 461.086,Z 514.784,A -85,B 0,C 180,E1 -8021.652,E2 -8021.652} C_VEL
LIN {X 0,Y 461.649,Z 504.943,A -85,B 0,C 180,E1 -8022.641,E2 -8022.641} C_VEL
LIN {X 0,Y 462.075,Z 494.066,A -85,B 0,C 180,E1 -8023.524,E2 -8023.524} C_VEL
LIN {X 0,Y 462.602,Z 481.862,A -85,B 0,C 180,E1 -8024.293,E2 -8024.293} C_VEL
LIN {X 0,Y 463.112,Z 469.094,A -85,B 0,C 180,E1 -8024.895,E2 -8024.895} C_VEL
LIN {X 0,Y 463.467,Z 456.391,A -85,B 0,C 180,E1 -8025.305,E2 -8025.305} C_VEL
LIN {X 0,Y 463.76,Z 438.424,A -85,B 0,C 180,E1 -8025.633,E2 -8025.633} C_VEL
LIN {X 0,Y 464.158,Z 362.581,A -85,B 0,C 180,E1 -8026.817,E2 -8026.817} C_VEL
LIN {X 0,Y 461.304,Z 344.315,A -85,B 0,C 180,E1 -8027.221,E2 -8027.221} C_VEL
LIN {X 0,Y 461.932,Z 328.645,A -85,B 0,C 180,E1 -8030.019,E2 -8030.019} C_VEL
LIN {X 0,Y 462.669,Z 313.27,A -85,B 0,C 180,E1 -8032.79,E2 -8032.79} C_VEL
LIN {X 0,Y 462.501,Z 308.172,A -85,B 0,C 180,E1 -8033.736,E2 -8033.736} C_VEL
LIN {X 0,Y 460.569,Z 298.117,A -85,B 0,C 180,E1 -8035.704,E2 -8035.704} C_VEL
LIN {X 0,Y 460.553,Z 298.115,A -85,B 0,C 180,E1 -8038.234,E2 -8038.234} C_VEL
LIN {X 0,Y 460.524,Z 298.116,A -85,B 0,C 180,E1 -8041.283,E2 -8041.283} C_VEL
LIN {X 0,Y 460.535,Z 298.115,A -85,B 0,C 180,E1 -8044.506,E2 -8044.506} C_VEL
LIN {X 0,Y 460.502,Z 298.12,A -85,B 0,C 180,E1 -8047.624,E2 -8047.624} C_VEL
LIN {X 0,Y 460.523,Z 298.115,A -85,B 0,C 180,E1 -8051.013,E2 -8051.013} C_VEL
LIN {X 0,Y 460.516,Z 298.121,A -85,B 0,C 180,E1 -8054.589,E2 -8054.589} C_VEL
LIN {X 0,Y 460.508,Z 298.118,A -85,B 0,C 180,E1 -8057.817,E2 -8057.817} C_VEL
LIN {X 0,Y 460.535,Z 298.116,A -85,B 0,C 180,E1 -8061.105,E2 -8061.105} C_VEL
LIN {X 0,Y 460.512,Z 298.122,A -85,B 0,C 180,E1 -8064.554,E2 -8064.554} C_VEL
LIN {X 0,Y 460.535,Z 298.113,A -85,B 0,C 180,E1 -8067.716,E2 -8067.716} C_VEL
LIN {X 0,Y 460.531,Z 298.119,A -85,B 0,C 180,E1 -8070.768,E2 -8070.768} C_VEL
LIN {X 0,Y 460.534,Z 298.115,A -85,B 0,C 180,E1 -8073.733,E2 -8073.733} C_VEL
LIN {X 0,Y 460.547,Z 298.113,A -85,B 0,C 180,E1 -8076.624,E2 -8076.624} C_VEL
LIN {X 0,Y 460.555,Z 298.118,A -85,B 0,C 180,E1 -8079.453,E2 -8079.453} C_VEL
LIN {X 0,Y 460.553,Z 298.111,A -85,B 0,C 180,E1 -8082.23,E2 -8082.23} C_VEL
LIN {X 0,Y 460.568,Z 298.111,A -85,B 0,C 180,E1 -8084.965,E2 -8084.965} C_VEL
LIN {X 0,Y 460.613,Z 298.104,A -85,B 0,C 180,E1 -8088.559,E2 -8088.559} C_VEL
LIN {X 0,Y 460.617,Z 298.105,A -85,B 0,C 180,E1 -8091.223,E2 -8091.223} C_VEL
LIN {X 0,Y 460.696,Z 298.102,A -85,B 0,C 180,E1 -8093.87,E2 -8093.87} C_VEL
LIN {X 0,Y 460.791,Z 298.083,A -85,B 0,C 180,E1 -8097.377,E2 -8097.377} C_VEL
LIN {X 0,Y 460.853,Z 298.081,A -85,B 0,C 180,E1 -8100,E2 -8100} C_VEL
LIN {X 0,Y 460.793,Z 298.084,A -85,B 0,C 180,E1 -8102.622,E2 -8102.622} C_VEL
LIN {X 0,Y 460.68,Z 298.101,A -85,B 0,C 180,E1 -8106.13,E2 -8106.13} C_VEL
LIN {X 0,Y 460.623,Z 298.106,A -85,B 0,C 180,E1 -8108.776,E2 -8108.776} C_VEL
LIN {X 0,Y 460.617,Z 298.11,A -85,B 0,C 180,E1 -8112.445,E2 -8112.445} C_VEL
LIN {X 0,Y 460.604,Z 298.105,A -85,B 0,C 180,E1 -8115.997,E2 -8115.997} C_VEL
LIN {X 0,Y 460.571,Z 298.109,A -85,B 0,C 180,E1 -8119.615,E2 -8119.615} C_VEL
LIN {X 0,Y 460.513,Z 298.118,A -85,B 0,C 180,E1 -8122.428,E2 -8122.428} C_VEL
LIN {X 0,Y 460.551,Z 298.112,A -85,B 0,C 180,E1 -8125.796,E2 -8125.796} C_VEL
LIN {X 0,Y 460.529,Z 298.114,A -85,B 0,C 180,E1 -8128.234,E2 -8128.234} C_VEL
LIN {X 0,Y 460.523,Z 298.124,A -85,B 0,C 180,E1 -8131.282,E2 -8131.282} C_VEL
LIN {X 0,Y 460.524,Z 298.115,A -85,B 0,C 180,E1 -8134.503,E2 -8134.503} C_VEL
LIN {X 0,Y 460.501,Z 298.126,A -85,B 0,C 180,E1 -8137.623,E2 -8137.623} C_VEL
LIN {X 0,Y 460.537,Z 298.114,A -85,B 0,C 180,E1 -8140.268,E2 -8140.268} C_VEL
LIN {X 0,Y 460.51,Z 298.12,A -85,B 0,C 180,E1 -8143.374,E2 -8143.374} C_VEL
LIN {X 0,Y 460.51,Z 298.117,A -85,B 0,C 180,E1 -8146.625,E2 -8146.625} C_VEL
LIN {X 0,Y 460.536,Z 298.118,A -85,B 0,C 180,E1 -8149.731,E2 -8149.731} C_VEL
LIN {X 0,Y 460.498,Z 298.121,A -85,B 0,C 180,E1 -8152.524,E2 -8152.524} C_VEL
LIN {X 0,Y 460.547,Z 298.113,A -85,B 0,C 180,E1 -8155.623,E2 -8155.623} C_VEL
LIN {X 0,Y 460.539,Z 298.116,A -85,B 0,C 180,E1 -8158.744,E2 -8158.744} C_VEL
LIN {X 0,Y 460.552,Z 298.117,A -85,B 0,C 180,E1 -8162.261,E2 -8162.261} C_VEL
LIN {X 0,Y 460.535,Z 298.121,A -85,B 0,C 180,E1 -8164.703,E2 -8164.703} C_VEL
LIN {X 0,Y 460.511,Z 298.116,A -85,B 0,C 180,E1 -8167.571,E2 -8167.571} C_VEL
LIN {X 0,Y 460.568,Z 298.112,A -85,B 0,C 180,E1 -8170.384,E2 -8170.384} C_VEL
LIN {X 0,Y 460.605,Z 298.104,A -85,B 0,C 180,E1 -8174.058,E2 -8174.058} C_VEL
LIN {X 0,Y 460.61,Z 298.106,A -85,B 0,C 180,E1 -8177.665,E2 -8177.665} C_VEL
LIN {X 0,Y 460.571,Z 298.112,A -85,B 0,C 180,E1 -8179.215,E2 -8179.215} C_VEL
LIN {X 0,Y 459.896,Z 298.199,A -85,B 0,C 180,E1 -8179.702,E2 -8179.702} C_VEL
LIN {X 0,Y 457.065,Z 298.553,A -85,B 0,C 180,E1 -8180.463,E2 -8180.463} C_VEL
LIN {X 0,Y 454.231,Z 298.908,A -85,B 0,C 180,E1 -8181.234,E2 -8181.234} C_VEL
LIN {X 0,Y 453.569,Z 298.987,A -85,B 0,C 180,E1 -8181.731,E2 -8181.731} C_VEL
LIN {X 0,Y 453.625,Z 299.085,A -85,B 0,C 180,E1 -8182.156,E2 -8182.156} C_VEL
LIN {X 0,Y 454.746,Z 305.569,A -85,B 0,C 180,E1 -8183.566,E2 -8183.566} C_VEL
LIN {X 0,Y 454.513,Z 318.548,A -85,B 0,C 180,E1 -8186.231,E2 -8186.231} C_VEL
LIN {X 0,Y 454.414,Z 320.444,A -85,B 0,C 180,E1 -8186.615,E2 -8186.615} C_VEL
LIN {X 0,Y 457.576,Z 336.912,A -85,B 0,C 180,E1 -8186.995,E2 -8186.995} C_VEL
LIN {X 0,Y 456.757,Z 428.153,A -85,B 0,C 180,E1 -8188.456,E2 -8188.456} C_VEL
LIN {X 0,Y 456.459,Z 440.378,A -85,B 0,C 180,E1 -8188.814,E2 -8188.814} C_VEL
LIN {X 0,Y 456.061,Z 453.652,A -85,B 0,C 180,E1 -8189.392,E2 -8189.392} C_VEL
LIN {X 0,Y 455.557,Z 465.633,A -85,B 0,C 180,E1 -8190.11,E2 -8190.11} C_VEL
LIN {X 0,Y 454.994,Z 477.058,A -85,B 0,C 180,E1 -8190.995,E2 -8190.995} C_VEL
LIN {X 0,Y 454.437,Z 487.366,A -85,B 0,C 180,E1 -8191.993,E2 -8191.993} C_VEL
LIN {X 0,Y 453.898,Z 496.654,A -85,B 0,C 180,E1 -8193.106,E2 -8193.106} C_VEL
LIN {X 0,Y 453.489,Z 505.626,A -85,B 0,C 180,E1 -8194.443,E2 -8194.443} C_VEL
LIN {X 0,Y 453.083,Z 512.892,A -85,B 0,C 180,E1 -8195.786,E2 -8195.786} C_VEL
LIN {X 0,Y 452.89,Z 518.702,A -85,B 0,C 180,E1 -8197.131,E2 -8197.131} C_VEL
LIN {X 0,Y 452.679,Z 523.293,A -85,B 0,C 180,E1 -8198.481,E2 -8198.481} C_VEL
LIN {X 0,Y 452.516,Z 526.79,A -85,B 0,C 180,E1 -8199.836,E2 -8199.836} C_VEL
LIN {X 0,Y 452.499,Z 528.53,A -85,B 0,C 180,E1 -8200.741,E2 -8200.741} C_VEL
LIN {X 0,Y 452.464,Z 530.156,A -85,B 0,C 180,E1 -8201.886,E2 -8201.886} C_VEL
LIN {X 0,Y 452.355,Z 531.287,A -85,B 0,C 180,E1 -8203.476,E2 -8203.476} C_VEL
LIN {X 0,Y 452.361,Z 531.351,A -85,B 0,C 180,E1 -8204.393,E2 -8204.393} C_VEL
LIN {X 0,Y 452.416,Z 530.833,A -85,B 0,C 180,E1 -8205.607,E2 -8205.607} C_VEL
LIN {X 0,Y 452.406,Z 529.048,A -85,B 0,C 180,E1 -8207.166,E2 -8207.166} C_VEL
LIN {X 0,Y 452.611,Z 526.051,A -85,B 0,C 180,E1 -8208.704,E2 -8208.704} C_VEL
LIN {X 0,Y 452.751,Z 522.617,A -85,B 0,C 180,E1 -8209.967,E2 -8209.967} C_VEL
LIN {X 0,Y 452.994,Z 517.411,A -85,B 0,C 180,E1 -8211.429,E2 -8211.429} C_VEL
LIN {X 0,Y 453.313,Z 511.17,A -85,B 0,C 180,E1 -8212.804,E2 -8212.804} C_VEL
LIN {X 0,Y 453.722,Z 504.269,A -85,B 0,C 180,E1 -8214.031,E2 -8214.031} C_VEL
LIN {X 0,Y 454.181,Z 496.391,A -85,B 0,C 180,E1 -8215.183,E2 -8215.183} C_VEL
LIN {X 0,Y 454.715,Z 486.085,A -85,B 0,C 180,E1 -8216.402,E2 -8216.402} C_VEL
LIN {X 0,Y 455.368,Z 474.939,A -85,B 0,C 180,E1 -8217.456,E2 -8217.456} C_VEL
LIN {X 0,Y 455.992,Z 463.713,A -85,B 0,C 180,E1 -8218.289,E2 -8218.289} C_VEL
LIN {X 0,Y 456.476,Z 451.107,A -85,B 0,C 180,E1 -8219.01,E2 -8219.01} C_VEL
LIN {X 0,Y 456.91,Z 438.013,A -85,B 0,C 180,E1 -8219.548,E2 -8219.548} C_VEL
LIN {X 0,Y 457.202,Z 425.516,A -85,B 0,C 180,E1 -8219.876,E2 -8219.876} C_VEL
LIN {X 0,Y 457.968,Z 336.354,A -85,B 0,C 180,E1 -8221.311,E2 -8221.311} C_VEL
LIN {X 0,Y 454.676,Z 320.29,A -85,B 0,C 180,E1 -8221.736,E2 -8221.736} C_VEL
LIN {X 0,Y 455.094,Z 308.707,A -85,B 0,C 180,E1 -8224.041,E2 -8224.041} C_VEL
LIN {X 0,Y 454.069,Z 301.937,A -85,B 0,C 180,E1 -8225.478,E2 -8225.478} C_VEL
LIN {X 0,Y 453.449,Z 299.004,A -85,B 0,C 180,E1 -8226.151,E2 -8226.151} C_VEL
LIN {X 0,Y 453.442,Z 299.002,A -85,B 0,C 180,E1 -8229.453,E2 -8229.453} C_VEL
LIN {X 0,Y 453.449,Z 298.998,A -85,B 0,C 180,E1 -8231.931,E2 -8231.931} C_VEL
LIN {X 0,Y 453.474,Z 298.999,A -85,B 0,C 180,E1 -8235.471,E2 -8235.471} C_VEL
LIN {X 0,Y 453.443,Z 298.998,A -85,B 0,C 180,E1 -8238.205,E2 -8238.205} C_VEL
LIN {X 0,Y 453.457,Z 298.999,A -85,B 0,C 180,E1 -8240.797,E2 -8240.797} C_VEL
LIN {X 0,Y 453.445,Z 299,A -85,B 0,C 180,E1 -8243.917,E2 -8243.917} C_VEL
LIN {X 0,Y 453.466,Z 298.989,A -85,B 0,C 180,E1 -8247.15,E2 -8247.15} C_VEL
LIN {X 0,Y 453.457,Z 298.994,A -85,B 0,C 180,E1 -8250.267,E2 -8250.267} C_VEL
LIN {X 0,Y 453.45,Z 299.001,A -85,B 0,C 180,E1 -8253.291,E2 -8253.291} C_VEL
LIN {X 0,Y 453.482,Z 298.995,A -85,B 0,C 180,E1 -8256.238,E2 -8256.238} C_VEL
LIN {X 0,Y 453.472,Z 298.994,A -85,B 0,C 180,E1 -8259.117,E2 -8259.117} C_VEL
LIN {X 0,Y 453.476,Z 298.995,A -85,B 0,C 180,E1 -8261.943,E2 -8261.943} C_VEL
LIN {X 0,Y 453.504,Z 298.99,A -85,B 0,C 180,E1 -8264.725,E2 -8264.725} C_VEL
LIN {X 0,Y 453.555,Z 298.98,A -85,B 0,C 180,E1 -8267.471,E2 -8267.471} C_VEL
LIN {X 0,Y 453.545,Z 298.979,A -85,B 0,C 180,E1 -8271.086,E2 -8271.086} C_VEL
LIN {X 0,Y 453.616,Z 298.977,A -85,B 0,C 180,E1 -8273.774,E2 -8273.774} C_VEL
LIN {X 0,Y 453.675,Z 298.964,A -85,B 0,C 180,E1 -8277.336,E2 -8277.336} C_VEL
LIN {X 0,Y 453.734,Z 298.964,A -85,B 0,C 180,E1 -8280,E2 -8280} C_VEL
LIN {X 0,Y 453.69,Z 298.967,A -85,B 0,C 180,E1 -8282.664,E2 -8282.664} C_VEL
LIN {X 0,Y 453.644,Z 298.975,A -85,B 0,C 180,E1 -8286.226,E2 -8286.226} C_VEL
LIN {X 0,Y 453.56,Z 298.986,A -85,B 0,C 180,E1 -8288.914,E2 -8288.914} C_VEL
LIN {X 0,Y 453.555,Z 298.985,A -85,B 0,C 180,E1 -8292.529,E2 -8292.529} C_VEL
LIN {X 0,Y 453.536,Z 298.985,A -85,B 0,C 180,E1 -8296.196,E2 -8296.196} C_VEL
LIN {X 0,Y 453.508,Z 298.99,A -85,B 0,C 180,E1 -8299.04,E2 -8299.04} C_VEL
LIN {X 0,Y 453.467,Z 298.992,A -85,B 0,C 180,E1 -8301.837,E2 -8301.837} C_VEL
LIN {X 0,Y 453.462,Z 298.996,A -85,B 0,C 180,E1 -8304.738,E2 -8304.738} C_VEL
LIN {X 0,Y 453.482,Z 298.991,A -85,B 0,C 180,E1 -8307.95,E2 -8307.95} C_VEL
LIN {X 0,Y 453.468,Z 298.996,A -85,B 0,C 180,E1 -8310.76,E2 -8310.76} C_VEL
LIN {X 0,Y 453.469,Z 298.997,A -85,B 0,C 180,E1 -8313.914,E2 -8313.914} C_VEL
LIN {X 0,Y 453.443,Z 299.001,A -85,B 0,C 180,E1 -8317.191,E2 -8317.191} C_VEL
LIN {X 0,Y 453.465,Z 298.997,A -85,B 0,C 180,E1 -8320.612,E2 -8320.612} C_VEL
LIN {X 0,Y 453.455,Z 298.997,A -85,B 0,C 180,E1 -8324.223,E2 -8324.223} C_VEL
LIN {X 0,Y 453.443,Z 299,A -85,B 0,C 180,E1 -8327.004,E2 -8327.004} C_VEL
LIN {X 0,Y 453.489,Z 298.997,A -85,B 0,C 180,E1 -8329.41,E2 -8329.41} C_VEL
LIN {X 0,Y 453.446,Z 298.999,A -85,B 0,C 180,E1 -8332.811,E2 -8332.811} C_VEL
LIN {X 0,Y 453.474,Z 298.998,A -85,B 0,C 180,E1 -8336.088,E2 -8336.088} C_VEL
LIN {X 0,Y 453.474,Z 298.998,A -85,B 0,C 180,E1 -8339.242,E2 -8339.242} C_VEL
LIN {X 0,Y 453.531,Z 298.993,A -85,B 0,C 180,E1 -8342.298,E2 -8342.298} C_VEL
LIN {X 0,Y 453.547,Z 299.158,A -85,B 0,C 180,E1 -8343.794,E2 -8343.794} C_VEL
LIN {X 0,Y 455.66,Z 309.861,A -85,B 0,C 180,E1 -8345.99,E2 -8345.99} C_VEL
LIN {X 0,Y 456.025,Z 314.323,A -85,B 0,C 180,E1 -8346.86,E2 -8346.86} C_VEL
LIN {X 0,Y 454.957,Z 333.699,A -85,B 0,C 180,E1 -8350.443,E2 -8350.443} C_VEL
LIN {X 0,Y 454.476,Z 343.956,A -85,B 0,C 180,E1 -8352.315,E2 -8352.315} C_VEL
LIN {X 0,Y 457.872,Z 364.691,A -85,B 0,C 180,E1 -8352.805,E2 -8352.805} C_VEL
LIN {X 0,Y 457.135,Z 452.226,A -85,B 0,C 180,E1 -8354.222,E2 -8354.222} C_VEL
LIN {X 0,Y 456.68,Z 464.673,A -85,B 0,C 180,E1 -8354.578,E2 -8354.578} C_VEL
LIN {X 0,Y 456.162,Z 478.11,A -85,B 0,C 180,E1 -8355.16,E2 -8355.16} C_VEL
LIN {X 0,Y 455.596,Z 489.407,A -85,B 0,C 180,E1 -8355.826,E2 -8355.826} C_VEL
LIN {X 0,Y 454.922,Z 501.179,A -85,B 0,C 180,E1 -8356.725,E2 -8356.725} C_VEL
LIN {X 0,Y 454.396,Z 511.573,A -85,B 0,C 180,E1 -8357.722,E2 -8357.722} C_VEL
LIN {X 0,Y 453.832,Z 521.047,A -85,B 0,C 180,E1 -8358.839,E2 -8358.839} C_VEL
LIN {X 0,Y 453.357,Z 530.178,A -85,B 0,C 180,E1 -8360.183,E2 -8360.183} C_VEL
LIN {X 0,Y 452.954,Z 537.543,A -85,B 0,C 180,E1 -8361.525,E2 -8361.525} C_VEL
LIN {X 0,Y 452.722,Z 543.461,A -85,B 0,C 180,E1 -8362.867,E2 -8362.867} C_VEL
LIN {X 0,Y 452.562,Z 548.136,A -85,B 0,C 180,E1 -8364.208,E2 -8364.208} C_VEL
LIN {X 0,Y 452.486,Z 551.706,A -85,B 0,C 180,E1 -8365.547,E2 -8365.547} C_VEL
LIN {X 0,Y 452.479,Z 553.538,A -85,B 0,C 180,E1 -8366.439,E2 -8366.439} C_VEL
LIN {X 0,Y 452.507,Z 554.916,A -85,B 0,C 180,E1 -8367.33,E2 -8367.33} C_VEL
LIN {X 0,Y 452.428,Z 556.492,A -85,B 0,C 180,E1 -8369.111,E2 -8369.111} C_VEL
LIN {X 0,Y 452.435,Z 556.684,A -85,B 0,C 180,E1 -8370.001,E2 -8370.001} C_VEL
LIN {X 0,Y 452.436,Z 555.825,A -85,B 0,C 180,E1 -8371.781,E2 -8371.781} C_VEL
LIN {X 0,Y 452.508,Z 554.815,A -85,B 0,C 180,E1 -8372.671,E2 -8372.671} C_VEL
LIN {X 0,Y 452.481,Z 553.386,A -85,B 0,C 180,E1 -8373.563,E2 -8373.563} C_VEL
LIN {X 0,Y 452.546,Z 550.413,A -85,B 0,C 180,E1 -8374.901,E2 -8374.901} C_VEL
LIN {X 0,Y 452.612,Z 545.827,A -85,B 0,C 180,E1 -8376.397,E2 -8376.397} C_VEL
LIN {X 0,Y 452.846,Z 539.167,A -85,B 0,C 180,E1 -8378.03,E2 -8378.03} C_VEL
LIN {X 0,Y 453.168,Z 532.167,A -85,B 0,C 180,E1 -8379.373,E2 -8379.373} C_VEL
LIN {X 0,Y 453.564,Z 523.381,A -85,B 0,C 180,E1 -8380.717,E2 -8380.717} C_VEL
LIN {X 0,Y 454.179,Z 513.405,A -85,B 0,C 180,E1 -8381.945,E2 -8381.945} C_VEL
LIN {X 0,Y 454.71,Z 502.657,A -85,B 0,C 180,E1 -8383.003,E2 -8383.003} C_VEL
LIN {X 0,Y 455.261,Z 491.955,A -85,B 0,C 180,E1 -8383.845,E2 -8383.845} C_VEL
LIN {X 0,Y 455.75,Z 480.258,A -85,B 0,C 180,E1 -8384.57,E2 -8384.57} C_VEL
LIN {X 0,Y 456.208,Z 467.586,A -85,B 0,C 180,E1 -8385.154,E2 -8385.154} C_VEL
LIN {X 0,Y 456.632,Z 454.121,A -85,B 0,C 180,E1 -8385.569,E2 -8385.569} C_VEL
LIN {X 0,Y 456.94,Z 427.822,A -85,B 0,C 180,E1 -8386.016,E2 -8386.016} C_VEL
LIN {X 0,Y 457.308,Z 363.418,A -85,B 0,C 180,E1 -8387.037,E2 -8387.037} C_VEL
LIN {X 0,Y 454.292,Z 344.131,A -85,B 0,C 180,E1 -8387.465,E2 -8387.465} C_VEL
LIN {X 0,Y 454.95,Z 329.567,A -85,B 0,C 180,E1 -8390.104,E2 -8390.104} C_VEL
LIN {X 0,Y 455.701,Z 314.189,A -85,B 0,C 180,E1 -8392.919,E2 -8392.919} C_VEL
LIN {X 0,Y 455.663,Z 310.32,A -85,B 0,C 180,E1 -8393.642,E2 -8393.642} C_VEL
LIN {X 0,Y 453.526,Z 298.995,A -85,B 0,C 180,E1 -8395.902,E2 -8395.902} C_VEL
LIN {X 0,Y 453.511,Z 298.99,A -85,B 0,C 180,E1 -8398.712,E2 -8398.712} C_VEL
LIN {X 0,Y 453.468,Z 299.001,A -85,B 0,C 180,E1 -8401.8,E2 -8401.8} C_VEL
LIN {X 0,Y 453.483,Z 298.992,A -85,B 0,C 180,E1 -8404.99,E2 -8404.99} C_VEL
LIN {X 0,Y 453.461,Z 299.001,A -85,B 0,C 180,E1 -8408.313,E2 -8408.313} C_VEL
LIN {X 0,Y 453.474,Z 298.996,A -85,B 0,C 180,E1 -8410.612,E2 -8410.612} C_VEL
LIN {X 0,Y 453.464,Z 299.001,A -85,B 0,C 180,E1 -8414.222,E2 -8414.222} C_VEL
LIN {X 0,Y 453.452,Z 298.997,A -85,B 0,C 180,E1 -8417.003,E2 -8417.003} C_VEL
LIN {X 0,Y 453.498,Z 298.99,A -85,B 0,C 180,E1 -8419.409,E2 -8419.409} C_VEL
LIN {X 0,Y 453.453,Z 299.002,A -85,B 0,C 180,E1 -8422.81,E2 -8422.81} C_VEL
LIN {X 0,Y 453.48,Z 298.993,A -85,B 0,C 180,E1 -8426.087,E2 -8426.087} C_VEL
LIN {X 0,Y 453.479,Z 298.997,A -85,B 0,C 180,E1 -8429.24,E2 -8429.24} C_VEL
LIN {X 0,Y 453.511,Z 298.989,A -85,B 0,C 180,E1 -8432.296,E2 -8432.296} C_VEL
LIN {X 0,Y 453.497,Z 298.997,A -85,B 0,C 180,E1 -8435.264,E2 -8435.264} C_VEL
LIN {X 0,Y 453.484,Z 298.992,A -85,B 0,C 180,E1 -8438.415,E2 -8438.415} C_VEL
LIN {X 0,Y 453.526,Z 298.99,A -85,B 0,C 180,E1 -8441.009,E2 -8441.009} C_VEL
LIN {X 0,Y 453.573,Z 298.984,A -85,B 0,C 180,E1 -8443.88,E2 -8443.88} C_VEL
LIN {X 0,Y 453.568,Z 298.988,A -85,B 0,C 180,E1 -8447.471,E2 -8447.471} C_VEL
LIN {X 0,Y 453.583,Z 298.98,A -85,B 0,C 180,E1 -8451.086,E2 -8451.086} C_VEL
LIN {X 0,Y 453.662,Z 298.977,A -85,B 0,C 180,E1 -8453.774,E2 -8453.774} C_VEL
LIN {X 0,Y 453.734,Z 298.961,A -85,B 0,C 180,E1 -8457.336,E2 -8457.336} C_VEL
LIN {X 0,Y 453.823,Z 298.957,A -85,B 0,C 180,E1 -8460,E2 -8460} C_VEL
LIN {X 0,Y 453.737,Z 298.963,A -85,B 0,C 180,E1 -8462.663,E2 -8462.663} C_VEL
LIN {X 0,Y 453.646,Z 298.978,A -85,B 0,C 180,E1 -8466.226,E2 -8466.226} C_VEL
LIN {X 0,Y 453.588,Z 298.981,A -85,B 0,C 180,E1 -8468.913,E2 -8468.913} C_VEL
LIN {X 0,Y 453.567,Z 298.989,A -85,B 0,C 180,E1 -8472.529,E2 -8472.529} C_VEL
LIN {X 0,Y 453.548,Z 298.986,A -85,B 0,C 180,E1 -8476.196,E2 -8476.196} C_VEL
LIN {X 0,Y 453.52,Z 298.993,A -85,B 0,C 180,E1 -8479.039,E2 -8479.039} C_VEL
LIN {X 0,Y 453.479,Z 298.992,A -85,B 0,C 180,E1 -8481.836,E2 -8481.836} C_VEL
LIN {X 0,Y 453.502,Z 298.994,A -85,B 0,C 180,E1 -8484.735,E2 -8484.735} C_VEL
LIN {X 0,Y 453.508,Z 298.989,A -85,B 0,C 180,E1 -8487.953,E2 -8487.953} C_VEL
LIN {X 0,Y 453.477,Z 298.994,A -85,B 0,C 180,E1 -8490.759,E2 -8490.759} C_VEL
LIN {X 0,Y 453.47,Z 298.996,A -85,B 0,C 180,E1 -8493.913,E2 -8493.913} C_VEL
LIN {X 0,Y 453.452,Z 299,A -85,B 0,C 180,E1 -8497.19,E2 -8497.19} C_VEL
LIN {X 0,Y 453.495,Z 298.99,A -85,B 0,C 180,E1 -8500.609,E2 -8500.609} C_VEL
LIN {X 0,Y 453.462,Z 298.997,A -85,B 0,C 180,E1 -8504.221,E2 -8504.221} C_VEL
LIN {X 0,Y 453.45,Z 298.996,A -85,B 0,C 180,E1 -8507.003,E2 -8507.003} C_VEL
LIN {X 0,Y 453.495,Z 298.992,A -85,B 0,C 180,E1 -8509.409,E2 -8509.409} C_VEL
LIN {X 0,Y 453.451,Z 298.997,A -85,B 0,C 180,E1 -8512.809,E2 -8512.809} C_VEL
LIN {X 0,Y 453.478,Z 298.999,A -85,B 0,C 180,E1 -8516.087,E2 -8516.087} C_VEL
LIN {X 0,Y 453.477,Z 298.993,A -85,B 0,C 180,E1 -8519.24,E2 -8519.24} C_VEL
LIN {X 0,Y 453.509,Z 298.994,A -85,B 0,C 180,E1 -8522.295,E2 -8522.295} C_VEL
LIN {X 0,Y 453.495,Z 298.991,A -85,B 0,C 180,E1 -8525.264,E2 -8525.264} C_VEL
LIN {X 0,Y 453.482,Z 298.996,A -85,B 0,C 180,E1 -8528.414,E2 -8528.414} C_VEL
LIN {X 0,Y 453.523,Z 298.993,A -85,B 0,C 180,E1 -8531.008,E2 -8531.008} C_VEL
LIN {X 0,Y 453.57,Z 298.981,A -85,B 0,C 180,E1 -8533.879,E2 -8533.879} C_VEL
LIN {X 0,Y 453.565,Z 298.985,A -85,B 0,C 180,E1 -8537.47,E2 -8537.47} C_VEL
LIN {X 0,Y 453.584,Z 298.988,A -85,B 0,C 180,E1 -8541.086,E2 -8541.086} C_VEL
LIN {X 0,Y 453.569,Z 298.987,A -85,B 0,C 180,E1 -8541.731,E2 -8541.731} C_VEL
LIN {X 0,Y 453.424,Z 299.516,A -85,B 0,C 180,E1 -8542.105,E2 -8542.105} C_VEL
LIN {X 0,Y 452.671,Z 301.78,A -85,B 0,C 180,E1 -8542.676,E2 -8542.676} C_VEL
LIN {X 0,Y 447.994,Z 312.664,A -85,B 0,C 180,E1 -8544.727,E2 -8544.727} C_VEL
LIN {X 0,Y 447.679,Z 314.737,A -85,B 0,C 180,E1 -8545.154,E2 -8545.154} C_VEL
LIN {X 0,Y 447.456,Z 320.641,A -85,B 0,C 180,E1 -8546.369,E2 -8546.369} C_VEL
LIN {X 0,Y 450.745,Z 338.194,A -85,B 0,C 180,E1 -8546.776,E2 -8546.776} C_VEL
LIN {X 0,Y 449.882,Z 428.165,A -85,B 0,C 180,E1 -8548.237,E2 -8548.237} C_VEL
LIN {X 0,Y 449.55,Z 440.475,A -85,B 0,C 180,E1 -8548.599,E2 -8548.599} C_VEL
LIN {X 0,Y 449.204,Z 453.199,A -85,B 0,C 180,E1 -8549.159,E2 -8549.159} C_VEL
LIN {X 0,Y 448.669,Z 465.388,A -85,B 0,C 180,E1 -8549.887,E2 -8549.887} C_VEL
LIN {X 0,Y 448.07,Z 476.908,A -85,B 0,C 180,E1 -8550.786,E2 -8550.786} C_VEL
LIN {X 0,Y 447.473,Z 487.289,A -85,B 0,C 180,E1 -8551.799,E2 -8551.799} C_VEL
LIN {X 0,Y 446.906,Z 496.648,A -85,B 0,C 180,E1 -8552.929,E2 -8552.929} C_VEL
LIN {X 0,Y 446.45,Z 505.667,A -85,B 0,C 180,E1 -8554.287,E2 -8554.287} C_VEL
LIN {X 0,Y 446.016,Z 512.962,A -85,B 0,C 180,E1 -8555.651,E2 -8555.651} C_VEL
LIN {X 0,Y 445.877,Z 517.838,A -85,B 0,C 180,E1 -8556.776,E2 -8556.776} C_VEL
LIN {X 0,Y 445.642,Z 522.695,A -85,B 0,C 180,E1 -8558.159,E2 -8558.159} C_VEL
LIN {X 0,Y 445.469,Z 526.389,A -85,B 0,C 180,E1 -8559.534,E2 -8559.534} C_VEL
LIN {X 0,Y 445.39,Z 529.054,A -85,B 0,C 180,E1 -8560.914,E2 -8560.914} C_VEL
LIN {X 0,Y 445.371,Z 530.43,A -85,B 0,C 180,E1 -8561.941,E2 -8561.941} C_VEL
LIN {X 0,Y 445.266,Z 531.522,A -85,B 0,C 180,E1 -8563.694,E2 -8563.694} C_VEL
LIN {X 0,Y 445.288,Z 531.514,A -85,B 0,C 180,E1 -8564.626,E2 -8564.626} C_VEL
LIN {X 0,Y 445.319,Z 530.993,A -85,B 0,C 180,E1 -8565.699,E2 -8565.699} C_VEL
LIN {X 0,Y 445.34,Z 528.916,A -85,B 0,C 180,E1 -8567.447,E2 -8567.447} C_VEL
LIN {X 0,Y 445.536,Z 526.171,A -85,B 0,C 180,E1 -8568.835,E2 -8568.835} C_VEL
LIN {X 0,Y 445.72,Z 522.157,A -85,B 0,C 180,E1 -8570.296,E2 -8570.296} C_VEL
LIN {X 0,Y 445.978,Z 516.632,A -85,B 0,C 180,E1 -8571.819,E2 -8571.819} C_VEL
LIN {X 0,Y 446.378,Z 510.309,A -85,B 0,C 180,E1 -8573.178,E2 -8573.178} C_VEL
LIN {X 0,Y 446.886,Z 501.843,A -85,B 0,C 180,E1 -8574.628,E2 -8574.628} C_VEL
LIN {X 0,Y 447.46,Z 493.089,A -85,B 0,C 180,E1 -8575.839,E2 -8575.839} C_VEL
LIN {X 0,Y 447.991,Z 483.894,A -85,B 0,C 180,E1 -8576.879,E2 -8576.879} C_VEL
LIN {X 0,Y 448.564,Z 474.104,A -85,B 0,C 180,E1 -8577.781,E2 -8577.781} C_VEL
LIN {X 0,Y 449.204,Z 463.21,A -85,B 0,C 180,E1 -8578.585,E2 -8578.585} C_VEL
LIN {X 0,Y 449.731,Z 450.802,A -85,B 0,C 180,E1 -8579.295,E2 -8579.295} C_VEL
LIN {X 0,Y 450.141,Z 438.359,A -85,B 0,C 180,E1 -8579.812,E2 -8579.812} C_VEL
LIN {X 0,Y 450.446,Z 425.971,A -85,B 0,C 180,E1 -8580.144,E2 -8580.144} C_VEL
LIN {X 0,Y 451.361,Z 337.803,A -85,B 0,C 180,E1 -8581.58,E2 -8581.58} C_VEL
LIN {X 0,Y 447.771,Z 320.477,A -85,B 0,C 180,E1 -8582.053,E2 -8582.053} C_VEL
LIN {X 0,Y 448.115,Z 309.023,A -85,B 0,C 180,E1 -8584.374,E2 -8584.374} C_VEL
LIN {X 0,Y 446.6,Z 300.799,A -85,B 0,C 180,E1 -8586.165,E2 -8586.165} C_VEL
LIN {X 0,Y 446.398,Z 299.883,A -85,B 0,C 180,E1 -8586.393,E2 -8586.393} C_VEL
LIN {X 0,Y 446.395,Z 299.879,A -85,B 0,C 180,E1 -8589.516,E2 -8589.516} C_VEL
LIN {X 0,Y 446.409,Z 299.878,A -85,B 0,C 180,E1 -8592.606,E2 -8592.606} C_VEL
LIN {X 0,Y 446.442,Z 299.877,A -85,B 0,C 180,E1 -8595.103,E2 -8595.103} C_VEL
LIN {X 0,Y 446.397,Z 299.877,A -85,B 0,C 180,E1 -8598.606,E2 -8598.606} C_VEL
LIN {X 0,Y 446.403,Z 299.876,A -85,B 0,C 180,E1 -8601.921,E2 -8601.921} C_VEL
LIN {X 0,Y 446.414,Z 299.868,A -85,B 0,C 180,E1 -8605.476,E2 -8605.476} C_VEL
LIN {X 0,Y 446.405,Z 299.876,A -85,B 0,C 180,E1 -8608.699,E2 -8608.699} C_VEL
LIN {X 0,Y 446.44,Z 299.876,A -85,B 0,C 180,E1 -8611.83,E2 -8611.83} C_VEL
LIN {X 0,Y 446.41,Z 299.872,A -85,B 0,C 180,E1 -8614.845,E2 -8614.845} C_VEL
LIN {X 0,Y 446.439,Z 299.871,A -85,B 0,C 180,E1 -8618.245,E2 -8618.245} C_VEL
LIN {X 0,Y 446.43,Z 299.874,A -85,B 0,C 180,E1 -8621.648,E2 -8621.648} C_VEL
LIN {X 0,Y 446.446,Z 299.871,A -85,B 0,C 180,E1 -8624.478,E2 -8624.478} C_VEL
LIN {X 0,Y 446.506,Z 299.857,A -85,B 0,C 180,E1 -8627.384,E2 -8627.384} C_VEL
LIN {X 0,Y 446.496,Z 299.858,A -85,B 0,C 180,E1 -8630.944,E2 -8630.944} C_VEL
LIN {X 0,Y 446.587,Z 299.852,A -85,B 0,C 180,E1 -8633.676,E2 -8633.676} C_VEL
LIN {X 0,Y 446.627,Z 299.842,A -85,B 0,C 180,E1 -8637.294,E2 -8637.294} C_VEL
LIN {X 0,Y 446.685,Z 299.843,A -85,B 0,C 180,E1 -8640,E2 -8640} C_VEL
LIN {X 0,Y 446.639,Z 299.845,A -85,B 0,C 180,E1 -8642.706,E2 -8642.706} C_VEL
LIN {X 0,Y 446.614,Z 299.852,A -85,B 0,C 180,E1 -8646.324,E2 -8646.324} C_VEL
LIN {X 0,Y 446.509,Z 299.864,A -85,B 0,C 180,E1 -8649.056,E2 -8649.056} C_VEL
LIN {X 0,Y 446.512,Z 299.86,A -85,B 0,C 180,E1 -8652.73,E2 -8652.73} C_VEL
LIN {X 0,Y 446.48,Z 299.866,A -85,B 0,C 180,E1 -8656.46,E2 -8656.46} C_VEL
LIN {X 0,Y 446.46,Z 299.87,A -85,B 0,C 180,E1 -8659.304,E2 -8659.304} C_VEL
LIN {X 0,Y 446.408,Z 299.871,A -85,B 0,C 180,E1 -8662.2,E2 -8662.2} C_VEL
LIN {X 0,Y 446.413,Z 299.879,A -85,B 0,C 180,E1 -8665.155,E2 -8665.155} C_VEL
LIN {X 0,Y 446.433,Z 299.869,A -85,B 0,C 180,E1 -8668.182,E2 -8668.182} C_VEL
LIN {X 0,Y 446.408,Z 299.877,A -85,B 0,C 180,E1 -8671.301,E2 -8671.301} C_VEL
LIN {X 0,Y 446.421,Z 299.872,A -85,B 0,C 180,E1 -8674.524,E2 -8674.524} C_VEL
LIN {X 0,Y 446.404,Z 299.875,A -85,B 0,C 180,E1 -8678.079,E2 -8678.079} C_VEL
LIN {X 0,Y 446.405,Z 299.88,A -85,B 0,C 180,E1 -8681.394,E2 -8681.394} C_VEL
LIN {X 0,Y 446.445,Z 299.87,A -85,B 0,C 180,E1 -8685.105,E2 -8685.105} C_VEL
LIN {X 0,Y 446.414,Z 299.878,A -85,B 0,C 180,E1 -8688.609,E2 -8688.609} C_VEL
LIN {X 0,Y 446.42,Z 299.876,A -85,B 0,C 180,E1 -8690.972,E2 -8690.972} C_VEL
LIN {X 0,Y 446.414,Z 299.877,A -85,B 0,C 180,E1 -8694.375,E2 -8694.375} C_VEL
LIN {X 0,Y 446.42,Z 299.877,A -85,B 0,C 180,E1 -8697.64,E2 -8697.64} C_VEL
LIN {X 0,Y 446.445,Z 299.876,A -85,B 0,C 180,E1 -8700.792,E2 -8700.792} C_VEL
LIN {X 0,Y 446.446,Z 299.88,A -85,B 0,C 180,E1 -8703.483,E2 -8703.483} C_VEL
LIN {X 0,Y 448.824,Z 311.788,A -85,B 0,C 180,E1 -8705.977,E2 -8705.977} C_VEL
LIN {X 0,Y 449.023,Z 316.845,A -85,B 0,C 180,E1 -8706.966,E2 -8706.966} C_VEL
LIN {X 0,Y 447.982,Z 335.168,A -85,B 0,C 180,E1 -8710.407,E2 -8710.407} C_VEL
LIN {X 0,Y 447.568,Z 343.938,A -85,B 0,C 180,E1 -8712.004,E2 -8712.004} C_VEL
LIN {X 0,Y 451.094,Z 365.095,A -85,B 0,C 180,E1 -8712.518,E2 -8712.518} C_VEL
LIN {X 0,Y 450.377,Z 452.053,A -85,B 0,C 180,E1 -8713.95,E2 -8713.95} C_VEL
LIN {X 0,Y 449.902,Z 464.489,A -85,B 0,C 180,E1 -8714.31,E2 -8714.31} C_VEL
LIN {X 0,Y 449.366,Z 477.36,A -85,B 0,C 180,E1 -8714.872,E2 -8714.872} C_VEL
LIN {X 0,Y 448.725,Z 489.611,A -85,B 0,C 180,E1 -8715.604,E2 -8715.604} C_VEL
LIN {X 0,Y 448.022,Z 501.258,A -85,B 0,C 180,E1 -8716.514,E2 -8716.514} C_VEL
LIN {X 0,Y 447.449,Z 511.615,A -85,B 0,C 180,E1 -8717.529,E2 -8717.529} C_VEL
LIN {X 0,Y 446.861,Z 521.027,A -85,B 0,C 180,E1 -8718.663,E2 -8718.663} C_VEL
LIN {X 0,Y 446.334,Z 530.111,A -85,B 0,C 180,E1 -8720.027,E2 -8720.027} C_VEL
LIN {X 0,Y 445.906,Z 537.448,A -85,B 0,C 180,E1 -8721.39,E2 -8721.39} C_VEL
LIN {X 0,Y 445.666,Z 543.347,A -85,B 0,C 180,E1 -8722.753,E2 -8722.753} C_VEL
LIN {X 0,Y 445.485,Z 547.445,A -85,B 0,C 180,E1 -8723.938,E2 -8723.938} C_VEL
LIN {X 0,Y 445.412,Z 551.557,A -85,B 0,C 180,E1 -8725.476,E2 -8725.476} C_VEL
LIN {X 0,Y 445.377,Z 553.373,A -85,B 0,C 180,E1 -8726.382,E2 -8726.382} C_VEL
LIN {X 0,Y 445.432,Z 554.744,A -85,B 0,C 180,E1 -8727.288,E2 -8727.288} C_VEL
LIN {X 0,Y 445.338,Z 556.305,A -85,B 0,C 180,E1 -8729.097,E2 -8729.097} C_VEL
LIN {X 0,Y 445.343,Z 556.482,A -85,B 0,C 180,E1 -8730.001,E2 -8730.001} C_VEL
LIN {X 0,Y 445.356,Z 555.607,A -85,B 0,C 180,E1 -8731.809,E2 -8731.809} C_VEL
LIN {X 0,Y 445.433,Z 554.589,A -85,B 0,C 180,E1 -8732.714,E2 -8732.714} C_VEL
LIN {X 0,Y 445.38,Z 553.143,A -85,B 0,C 180,E1 -8733.62,E2 -8733.62} C_VEL
LIN {X 0,Y 445.474,Z 550.157,A -85,B 0,C 180,E1 -8734.979,E2 -8734.979} C_VEL
LIN {X 0,Y 445.558,Z 544.651,A -85,B 0,C 180,E1 -8736.749,E2 -8736.749} C_VEL
LIN {X 0,Y 445.787,Z 538.866,A -85,B 0,C 180,E1 -8738.158,E2 -8738.158} C_VEL
LIN {X 0,Y 446.127,Z 531.835,A -85,B 0,C 180,E1 -8739.522,E2 -8739.522} C_VEL
LIN {X 0,Y 446.555,Z 523.017,A -85,B 0,C 180,E1 -8740.887,E2 -8740.887} C_VEL
LIN {X 0,Y 447.187,Z 513.005,A -85,B 0,C 180,E1 -8742.135,E2 -8742.135} C_VEL
LIN {X 0,Y 447.727,Z 502.186,A -85,B 0,C 180,E1 -8743.209,E2 -8743.209} C_VEL
LIN {X 0,Y 448.323,Z 491.412,A -85,B 0,C 180,E1 -8744.063,E2 -8744.063} C_VEL
LIN {X 0,Y 448.87,Z 479.613,A -85,B 0,C 180,E1 -8744.798,E2 -8744.798} C_VEL
LIN {X 0,Y 449.32,Z 466.68,A -85,B 0,C 180,E1 -8745.392,E2 -8745.392} C_VEL
LIN {X 0,Y 449.75,Z 453.993,A -85,B 0,C 180,E1 -8745.784,E2 -8745.784} C_VEL
LIN {X 0,Y 450.097,Z 429.509,A -85,B 0,C 180,E1 -8746.208,E2 -8746.208} C_VEL
LIN {X 0,Y 450.47,Z 364.434,A -85,B 0,C 180,E1 -8747.254,E2 -8747.254} C_VEL
LIN {X 0,Y 447.302,Z 343.991,A -85,B 0,C 180,E1 -8747.707,E2 -8747.707} C_VEL
LIN {X 0,Y 448.001,Z 329.2,A -85,B 0,C 180,E1 -8750.43,E2 -8750.43} C_VEL
LIN {X 0,Y 448.791,Z 313.794,A -85,B 0,C 180,E1 -8753.292,E2 -8753.292} C_VEL
LIN {X 0,Y 448.086,Z 308.364,A -85,B 0,C 180,E1 -8754.356,E2 -8754.356} C_VEL
LIN {X 0,Y 446.464,Z 299.874,A -85,B 0,C 180,E1 -8756.103,E2 -8756.103} C_VEL
LIN {X 0,Y 446.451,Z 299.871,A -85,B 0,C 180,E1 -8759.21,E2 -8759.21} C_VEL
LIN {X 0,Y 446.427,Z 299.873,A -85,B 0,C 180,E1 -8762.362,E2 -8762.362} C_VEL
LIN {X 0,Y 446.422,Z 299.875,A -85,B 0,C 180,E1 -8765.627,E2 -8765.627} C_VEL
LIN {X 0,Y 446.411,Z 299.873,A -85,B 0,C 180,E1 -8769.031,E2 -8769.031} C_VEL
LIN {X 0,Y 446.423,Z 299.88,A -85,B 0,C 180,E1 -8772.275,E2 -8772.275} C_VEL
LIN {X 0,Y 446.454,Z 299.868,A -85,B 0,C 180,E1 -8775.104,E2 -8775.104} C_VEL
LIN {X 0,Y 446.423,Z 299.879,A -85,B 0,C 180,E1 -8778.608,E2 -8778.608} C_VEL
LIN {X 0,Y 446.428,Z 299.874,A -85,B 0,C 180,E1 -8780.971,E2 -8780.971} C_VEL
LIN {X 0,Y 446.421,Z 299.875,A -85,B 0,C 180,E1 -8784.374,E2 -8784.374} C_VEL
LIN {X 0,Y 446.425,Z 299.871,A -85,B 0,C 180,E1 -8787.638,E2 -8787.638} C_VEL
LIN {X 0,Y 446.441,Z 299.875,A -85,B 0,C 180,E1 -8790.79,E2 -8790.79} C_VEL
LIN {X 0,Y 446.442,Z 299.869,A -85,B 0,C 180,E1 -8793.846,E2 -8793.846} C_VEL
LIN {X 0,Y 446.428,Z 299.874,A -85,B 0,C 180,E1 -8796.823,E2 -8796.823} C_VEL
LIN {X 0,Y 446.448,Z 299.871,A -85,B 0,C 180,E1 -8799.737,E2 -8799.737} C_VEL
LIN {X 0,Y 446.46,Z 299.867,A -85,B 0,C 180,E1 -8802.597,E2 -8802.597} C_VEL
LIN {X 0,Y 446.473,Z 299.872,A -85,B 0,C 180,E1 -8805.412,E2 -8805.412} C_VEL
LIN {X 0,Y 446.521,Z 299.861,A -85,B 0,C 180,E1 -8808.193,E2 -8808.193} C_VEL
LIN {X 0,Y 446.531,Z 299.858,A -85,B 0,C 180,E1 -8810.944,E2 -8810.944} C_VEL
LIN {X 0,Y 446.631,Z 299.851,A -85,B 0,C 180,E1 -8813.676,E2 -8813.676} C_VEL
LIN {X 0,Y 446.681,Z 299.84,A -85,B 0,C 180,E1 -8817.294,E2 -8817.294} C_VEL
LIN {X 0,Y 446.792,Z 299.832,A -85,B 0,C 180,E1 -8820,E2 -8820} C_VEL
LIN {X 0,Y 446.684,Z 299.841,A -85,B 0,C 180,E1 -8822.705,E2 -8822.705} C_VEL
LIN {X 0,Y 446.615,Z 299.856,A -85,B 0,C 180,E1 -8826.324,E2 -8826.324} C_VEL
LIN {X 0,Y 446.536,Z 299.859,A -85,B 0,C 180,E1 -8829.055,E2 -8829.055} C_VEL
LIN {X 0,Y 446.525,Z 299.865,A -85,B 0,C 180,E1 -8832.729,E2 -8832.729} C_VEL
LIN {X 0,Y 446.499,Z 299.864,A -85,B 0,C 180,E1 -8836.227,E2 -8836.227} C_VEL
LIN {X 0,Y 446.471,Z 299.868,A -85,B 0,C 180,E1 -8839.303,E2 -8839.303} C_VEL
LIN {X 0,Y 446.42,Z 299.872,A -85,B 0,C 180,E1 -8842.199,E2 -8842.199} C_VEL
LIN {X 0,Y 446.445,Z 299.876,A -85,B 0,C 180,E1 -8845.153,E2 -8845.153} C_VEL
LIN {X 0,Y 446.451,Z 299.868,A -85,B 0,C 180,E1 -8848.181,E2 -8848.181} C_VEL
LIN {X 0,Y 446.418,Z 299.881,A -85,B 0,C 180,E1 -8851.3,E2 -8851.3} C_VEL
LIN {X 0,Y 446.424,Z 299.871,A -85,B 0,C 180,E1 -8854.523,E2 -8854.523} C_VEL
LIN {X 0,Y 446.413,Z 299.875,A -85,B 0,C 180,E1 -8858.078,E2 -8858.078} C_VEL
LIN {X 0,Y 446.424,Z 299.872,A -85,B 0,C 180,E1 -8860.916,E2 -8860.916} C_VEL
LIN {X 0,Y 446.401,Z 299.882,A -85,B 0,C 180,E1 -8863.846,E2 -8863.846} C_VEL
LIN {X 0,Y 446.399,Z 299.876,A -85,B 0,C 180,E1 -8866.403,E2 -8866.403} C_VEL
LIN {X 0,Y 446.434,Z 299.875,A -85,B 0,C 180,E1 -8869.8,E2 -8869.8} C_VEL
LIN {X 0,Y 446.401,Z 299.874,A -85,B 0,C 180,E1 -8873.254,E2 -8873.254} C_VEL
LIN {X 0,Y 446.45,Z 299.872,A -85,B 0,C 180,E1 -8876.566,E2 -8876.566} C_VEL
LIN {X 0,Y 446.43,Z 299.873,A -85,B 0,C 180,E1 -8879.979,E2 -8879.979} C_VEL
LIN {X 0,Y 446.446,Z 299.873,A -85,B 0,C 180,E1 -8882.836,E2 -8882.836} C_VEL
LIN {X 0,Y 446.461,Z 299.867,A -85,B 0,C 180,E1 -8885.924,E2 -8885.924} C_VEL
LIN {X 0,Y 446.454,Z 299.876,A -85,B 0,C 180,E1 -8888.772,E2 -8888.772} C_VEL
LIN {X 0,Y 446.451,Z 299.868,A -85,B 0,C 180,E1 -8891.648,E2 -8891.648} C_VEL
LIN {X 0,Y 446.508,Z 299.863,A -85,B 0,C 180,E1 -8894.479,E2 -8894.479} C_VEL
LIN {X 0,Y 446.517,Z 299.86,A -85,B 0,C 180,E1 -8898.192,E2 -8898.192} C_VEL
LIN {X 0,Y 446.531,Z 299.864,A -85,B 0,C 180,E1 -8900.944,E2 -8900.944} C_VEL
LIN {X 0,Y 446.55,Z 299.905,A -85,B 0,C 180,E1 -8901.979,E2 -8901.979} C_VEL
LIN {X 0,Y 447.748,Z 307.741,A -85,B 0,C 180,E1 -8903.691,E2 -8903.691} C_VEL
LIN {X 0,Y 447.679,Z 314.737,A -85,B 0,C 180,E1 -8905.154,E2 -8905.154} C_VEL
LIN {X 0,Y 447.464,Z 317.181,A -85,B 0,C 180,E1 -8905.534,E2 -8905.534} C_VEL
LIN {X 0,Y 447.014,Z 320.218,A -85,B 0,C 180,E1 -8905.837,E2 -8905.837} C_VEL
LIN {X 0,Y 446.095,Z 325.452,A -85,B 0,C 180,E1 -8906.165,E2 -8906.165} C_VEL
LIN {X 0,Y 445.087,Z 331.254,A -85,B 0,C 180,E1 -8906.376,E2 -8906.376} C_VEL
LIN {X 0,Y 444.492,Z 335.288,A -85,B 0,C 180,E1 -8906.473,E2 -8906.473} C_VEL
LIN {X 0,Y 443.887,Z 343.482,A -85,B 0,C 180,E1 -8906.617,E2 -8906.617} C_VEL
LIN {X 0,Y 443.003,Z 428.688,A -85,B 0,C 180,E1 -8908.025,E2 -8908.025} C_VEL
LIN {X 0,Y 442.666,Z 441.248,A -85,B 0,C 180,E1 -8908.407,E2 -8908.407} C_VEL
LIN {X 0,Y 442.291,Z 453.831,A -85,B 0,C 180,E1 -8908.975,E2 -8908.975} C_VEL
LIN {X 0,Y 441.776,Z 465.098,A -85,B 0,C 180,E1 -8909.657,E2 -8909.657} C_VEL
LIN {X 0,Y 441.149,Z 476.712,A -85,B 0,C 180,E1 -8910.57,E2 -8910.57} C_VEL
LIN {X 0,Y 440.508,Z 487.165,A -85,B 0,C 180,E1 -8911.599,E2 -8911.599} C_VEL
LIN {X 0,Y 439.944,Z 496.588,A -85,B 0,C 180,E1 -8912.746,E2 -8912.746} C_VEL
LIN {X 0,Y 439.412,Z 505.664,A -85,B 0,C 180,E1 -8914.126,E2 -8914.126} C_VEL
LIN {X 0,Y 438.954,Z 512.999,A -85,B 0,C 180,E1 -8915.512,E2 -8915.512} C_VEL
LIN {X 0,Y 438.738,Z 519.475,A -85,B 0,C 180,E1 -8917.064,E2 -8917.064} C_VEL
LIN {X 0,Y 438.451,Z 524.789,A -85,B 0,C 180,E1 -8918.758,E2 -8918.758} C_VEL
LIN {X 0,Y 438.33,Z 527.983,A -85,B 0,C 180,E1 -8920.157,E2 -8920.157} C_VEL
LIN {X 0,Y 438.289,Z 529.572,A -85,B 0,C 180,E1 -8921.093,E2 -8921.093} C_VEL
LIN {X 0,Y 438.275,Z 530.72,A -85,B 0,C 180,E1 -8922.031,E2 -8922.031} C_VEL
LIN {X 0,Y 438.197,Z 531.438,A -85,B 0,C 180,E1 -8922.975,E2 -8922.975} C_VEL
LIN {X 0,Y 438.166,Z 531.758,A -85,B 0,C 180,E1 -8923.921,E2 -8923.921} C_VEL
LIN {X 0,Y 438.203,Z 531.676,A -85,B 0,C 180,E1 -8924.868,E2 -8924.868} C_VEL
LIN {X 0,Y 438.236,Z 531.135,A -85,B 0,C 180,E1 -8925.82,E2 -8925.82} C_VEL
LIN {X 0,Y 438.214,Z 530.173,A -85,B 0,C 180,E1 -8926.778,E2 -8926.778} C_VEL
LIN {X 0,Y 438.285,Z 528.792,A -85,B 0,C 180,E1 -8927.737,E2 -8927.737} C_VEL
LIN {X 0,Y 438.475,Z 526.297,A -85,B 0,C 180,E1 -8928.974,E2 -8928.974} C_VEL
LIN {X 0,Y 438.697,Z 521.718,A -85,B 0,C 180,E1 -8930.636,E2 -8930.636} C_VEL
LIN {X 0,Y 439.079,Z 515.297,A -85,B 0,C 180,E1 -8932.332,E2 -8932.332} C_VEL
LIN {X 0,Y 439.558,Z 508.241,A -85,B 0,C 180,E1 -8933.783,E2 -8933.783} C_VEL
LIN {X 0,Y 440.04,Z 500.695,A -85,B 0,C 180,E1 -8935.038,E2 -8935.038} C_VEL
LIN {X 0,Y 440.648,Z 491.575,A -85,B 0,C 180,E1 -8936.268,E2 -8936.268} C_VEL
LIN {X 0,Y 441.321,Z 481.337,A -85,B 0,C 180,E1 -8937.385,E2 -8937.385} C_VEL
LIN {X 0,Y 442.027,Z 470.209,A -85,B 0,C 180,E1 -8938.358,E2 -8938.358} C_VEL
LIN {X 0,Y 442.658,Z 458.329,A -85,B 0,C 180,E1 -8939.165,E2 -8939.165} C_VEL
LIN {X 0,Y 443.14,Z 446.519,A -85,B 0,C 180,E1 -8939.774,E2 -8939.774} C_VEL
LIN {X 0,Y 443.511,Z 433.912,A -85,B 0,C 180,E1 -8940.238,E2 -8940.238} C_VEL
LIN {X 0,Y 443.763,Z 420.092,A -85,B 0,C 180,E1 -8940.541,E2 -8940.541} C_VEL
LIN {X 0,Y 444.634,Z 338.665,A -85,B 0,C 180,E1 -8941.88,E2 -8941.88} C_VEL
LIN {X 0,Y 440.906,Z 320.636,A -85,B 0,C 180,E1 -8942.39,E2 -8942.39} C_VEL
LIN {X 0,Y 441.211,Z 310.467,A -85,B 0,C 180,E1 -8944.479,E2 -8944.479} C_VEL
LIN {X 0,Y 439.716,Z 302.462,A -85,B 0,C 180,E1 -8946.253,E2 -8946.253} C_VEL
LIN {X 0,Y 439.351,Z 300.76,A -85,B 0,C 180,E1 -8946.663,E2 -8946.663} C_VEL
LIN {X 0,Y 439.341,Z 300.758,A -85,B 0,C 180,E1 -8949.84,E2 -8949.84} C_VEL
LIN {X 0,Y 439.363,Z 300.756,A -85,B 0,C 180,E1 -8952.624,E2 -8952.624} C_VEL
LIN {X 0,Y 439.39,Z 300.756,A -85,B 0,C 180,E1 -8955.27,E2 -8955.27} C_VEL
LIN {X 0,Y 439.348,Z 300.76,A -85,B 0,C 180,E1 -8959.016,E2 -8959.016} C_VEL
LIN {X 0,Y 439.359,Z 300.756,A -85,B 0,C 180,E1 -8961.608,E2 -8961.608} C_VEL
LIN {X 0,Y 439.388,Z 300.752,A -85,B 0,C 180,E1 -8964.843,E2 -8964.843} C_VEL
LIN {X 0,Y 439.36,Z 300.754,A -85,B 0,C 180,E1 -8968.139,E2 -8968.139} C_VEL
LIN {X 0,Y 439.394,Z 300.753,A -85,B 0,C 180,E1 -8971.605,E2 -8971.605} C_VEL
LIN {X 0,Y 439.355,Z 300.751,A -85,B 0,C 180,E1 -8974.412,E2 -8974.412} C_VEL
LIN {X 0,Y 439.354,Z 300.757,A -85,B 0,C 180,E1 -8977.424,E2 -8977.424} C_VEL
LIN {X 0,Y 439.431,Z 300.743,A -85,B 0,C 180,E1 -8980.663,E2 -8980.663} C_VEL
LIN {X 0,Y 439.407,Z 300.75,A -85,B 0,C 180,E1 -8984.223,E2 -8984.223} C_VEL
LIN {X 0,Y 439.474,Z 300.733,A -85,B 0,C 180,E1 -8987.286,E2 -8987.286} C_VEL
LIN {X 0,Y 439.462,Z 300.734,A -85,B 0,C 180,E1 -8990.798,E2 -8990.798} C_VEL
LIN {X 0,Y 439.539,Z 300.729,A -85,B 0,C 180,E1 -8993.574,E2 -8993.574} C_VEL
LIN {X 0,Y 439.39,Z 300.746,A -85,B 0,C 180,E1 -8995.413,E2 -8995.413} C_VEL
LIN {X 0,Y 439.614,Z 300.72,A -85,B 0,C 180,E1 -8998.168,E2 -8998.168} C_VEL
LIN {X 0,Y 439.574,Z 300.724,A -85,B 0,C 180,E1 -9000.916,E2 -9000.916} C_VEL
LIN {X 0,Y 439.591,Z 300.723,A -85,B 0,C 180,E1 -9002.749,E2 -9002.749} C_VEL
LIN {X 0,Y 439.585,Z 300.729,A -85,B 0,C 180,E1 -9006.426,E2 -9006.426} C_VEL
LIN {X 0,Y 439.473,Z 300.739,A -85,B 0,C 180,E1 -9009.202,E2 -9009.202} C_VEL
LIN {X 0,Y 439.456,Z 300.737,A -85,B 0,C 180,E1 -9012.938,E2 -9012.938} C_VEL
LIN {X 0,Y 439.438,Z 300.742,A -85,B 0,C 180,E1 -9016.348,E2 -9016.348} C_VEL
LIN {X 0,Y 439.394,Z 300.747,A -85,B 0,C 180,E1 -9019.627,E2 -9019.627} C_VEL
LIN {X 0,Y 439.354,Z 300.751,A -85,B 0,C 180,E1 -9022.576,E2 -9022.576} C_VEL
LIN {X 0,Y 439.358,Z 300.755,A -85,B 0,C 180,E1 -9025.588,E2 -9025.588} C_VEL
LIN {X 0,Y 439.389,Z 300.747,A -85,B 0,C 180,E1 -9028.676,E2 -9028.676} C_VEL
LIN {X 0,Y 439.362,Z 300.751,A -85,B 0,C 180,E1 -9032.031,E2 -9032.031} C_VEL
LIN {X 0,Y 439.387,Z 300.752,A -85,B 0,C 180,E1 -9035.341,E2 -9035.341} C_VEL
LIN {X 0,Y 439.356,Z 300.751,A -85,B 0,C 180,E1 -9038.598,E2 -9038.598} C_VEL
LIN {X 0,Y 439.365,Z 300.756,A -85,B 0,C 180,E1 -9041.255,E2 -9041.255} C_VEL
LIN {X 0,Y 439.393,Z 300.748,A -85,B 0,C 180,E1 -9044.731,E2 -9044.731} C_VEL
LIN {X 0,Y 439.38,Z 300.757,A -85,B 0,C 180,E1 -9047.795,E2 -9047.795} C_VEL
LIN {X 0,Y 439.385,Z 300.757,A -85,B 0,C 180,E1 -9050.224,E2 -9050.224} C_VEL
LIN {X 0,Y 439.369,Z 300.756,A -85,B 0,C 180,E1 -9053.714,E2 -9053.714} C_VEL
LIN {X 0,Y 439.37,Z 300.754,A -85,B 0,C 180,E1 -9057.055,E2 -9057.055} C_VEL
LIN {X 0,Y 439.379,Z 300.754,A -85,B 0,C 180,E1 -9060.275,E2 -9060.275} C_VEL
LIN {X 0,Y 439.43,Z 300.799,A -85,B 0,C 180,E1 -9063.205,E2 -9063.205} C_VEL
LIN {X 0,Y 441.879,Z 313.077,A -85,B 0,C 180,E1 -9065.825,E2 -9065.825} C_VEL
LIN {X 0,Y 442.215,Z 316.858,A -85,B 0,C 180,E1 -9066.59,E2 -9066.59} C_VEL
LIN {X 0,Y 441.111,Z 334.988,A -85,B 0,C 180,E1 -9070.055,E2 -9070.055} C_VEL
LIN {X 0,Y 440.637,Z 343.503,A -85,B 0,C 180,E1 -9071.663,E2 -9071.663} C_VEL
LIN {X 0,Y 443.843,Z 362.115,A -85,B 0,C 180,E1 -9072.138,E2 -9072.138} C_VEL
LIN {X 0,Y 444.449,Z 367.924,A -85,B 0,C 180,E1 -9072.265,E2 -9072.265} C_VEL
LIN {X 0,Y 443.635,Z 451.884,A -85,B 0,C 180,E1 -9073.67,E2 -9073.67} C_VEL
LIN {X 0,Y 443.143,Z 464.305,A -85,B 0,C 180,E1 -9074.035,E2 -9074.035} C_VEL
LIN {X 0,Y 442.542,Z 477.733,A -85,B 0,C 180,E1 -9074.633,E2 -9074.633} C_VEL
LIN {X 0,Y 441.872,Z 489.812,A -85,B 0,C 180,E1 -9075.376,E2 -9075.376} C_VEL
LIN {X 0,Y 441.095,Z 501.588,A -85,B 0,C 180,E1 -9076.316,E2 -9076.316} C_VEL
LIN {X 0,Y 440.514,Z 511.687,A -85,B 0,C 180,E1 -9077.329,E2 -9077.329} C_VEL
LIN {X 0,Y 439.899,Z 521.036,A -85,B 0,C 180,E1 -9078.481,E2 -9078.481} C_VEL
LIN {X 0,Y 439.321,Z 530.083,A -85,B 0,C 180,E1 -9079.866,E2 -9079.866} C_VEL
LIN {X 0,Y 438.864,Z 537.387,A -85,B 0,C 180,E1 -9081.25,E2 -9081.25} C_VEL
LIN {X 0,Y 438.603,Z 543.253,A -85,B 0,C 180,E1 -9082.636,E2 -9082.636} C_VEL
LIN {X 0,Y 438.386,Z 547.756,A -85,B 0,C 180,E1 -9083.978,E2 -9083.978} C_VEL
LIN {X 0,Y 438.341,Z 551.415,A -85,B 0,C 180,E1 -9085.403,E2 -9085.403} C_VEL
LIN {X 0,Y 438.279,Z 553.211,A -85,B 0,C 180,E1 -9086.323,E2 -9086.323} C_VEL
LIN {X 0,Y 438.34,Z 554.573,A -85,B 0,C 180,E1 -9087.244,E2 -9087.244} C_VEL
LIN {X 0,Y 438.252,Z 556.119,A -85,B 0,C 180,E1 -9089.082,E2 -9089.082} C_VEL
LIN {X 0,Y 438.254,Z 556.279,A -85,B 0,C 180,E1 -9090.001,E2 -9090.001} C_VEL
LIN {X 0,Y 438.278,Z 555.39,A -85,B 0,C 180,E1 -9091.839,E2 -9091.839} C_VEL
LIN {X 0,Y 438.341,Z 554.363,A -85,B 0,C 180,E1 -9092.758,E2 -9092.758} C_VEL
LIN {X 0,Y 438.281,Z 552.899,A -85,B 0,C 180,E1 -9093.678,E2 -9093.678} C_VEL
LIN {X 0,Y 438.384,Z 549.896,A -85,B 0,C 180,E1 -9095.059,E2 -9095.059} C_VEL
LIN {X 0,Y 438.449,Z 545.827,A -85,B 0,C 180,E1 -9096.443,E2 -9096.443} C_VEL
LIN {X 0,Y 438.683,Z 539.568,A -85,B 0,C 180,E1 -9098.059,E2 -9098.059} C_VEL
LIN {X 0,Y 439.014,Z 532.748,A -85,B 0,C 180,E1 -9099.445,E2 -9099.445} C_VEL
LIN {X 0,Y 439.441,Z 524.252,A -85,B 0,C 180,E1 -9100.832,E2 -9100.832} C_VEL
LIN {X 0,Y 440.006,Z 515.498,A -85,B 0,C 180,E1 -9101.985,E2 -9101.985} C_VEL
LIN {X 0,Y 440.604,Z 505.459,A -85,B 0,C 180,E1 -9103.065,E2 -9103.065} C_VEL
LIN {X 0,Y 441.13,Z 495.404,A -85,B 0,C 180,E1 -9103.944,E2 -9103.944} C_VEL
LIN {X 0,Y 441.729,Z 483.862,A -85,B 0,C 180,E1 -9104.748,E2 -9104.748} C_VEL
LIN {X 0,Y 442.275,Z 471.889,A -85,B 0,C 180,E1 -9105.378,E2 -9105.378} C_VEL
LIN {X 0,Y 442.749,Z 459.874,A -85,B 0,C 180,E1 -9105.833,E2 -9105.833} C_VEL
LIN {X 0,Y 443.042,Z 446.912,A -85,B 0,C 180,E1 -9106.148,E2 -9106.148} C_VEL
LIN {X 0,Y 443.63,Z 365.307,A -85,B 0,C 180,E1 -9107.479,E2 -9107.479} C_VEL
LIN {X 0,Y 440.337,Z 343.71,A -85,B 0,C 180,E1 -9107.978,E2 -9107.978} C_VEL
LIN {X 0,Y 441.18,Z 327.525,A -85,B 0,C 180,E1 -9111.004,E2 -9111.004} C_VEL
LIN {X 0,Y 441.828,Z 314.676,A -85,B 0,C 180,E1 -9113.433,E2 -9113.433} C_VEL
LIN {X 0,Y 440.884,Z 308.432,A -85,B 0,C 180,E1 -9114.684,E2 -9114.684} C_VEL
LIN {X 0,Y 439.429,Z 300.749,A -85,B 0,C 180,E1 -9116.281,E2 -9116.281} C_VEL
LIN {X 0,Y 439.421,Z 300.746,A -85,B 0,C 180,E1 -9118.674,E2 -9118.674} C_VEL
LIN {X 0,Y 439.375,Z 300.756,A -85,B 0,C 180,E1 -9122.031,E2 -9122.031} C_VEL
LIN {X 0,Y 439.397,Z 300.747,A -85,B 0,C 180,E1 -9125.34,E2 -9125.34} C_VEL
LIN {X 0,Y 439.366,Z 300.753,A -85,B 0,C 180,E1 -9128.597,E2 -9128.597} C_VEL
LIN {X 0,Y 439.386,Z 300.756,A -85,B 0,C 180,E1 -9132.206,E2 -9132.206} C_VEL
LIN {X 0,Y 439.403,Z 300.746,A -85,B 0,C 180,E1 -9135.271,E2 -9135.271} C_VEL
LIN {X 0,Y 439.385,Z 300.753,A -85,B 0,C 180,E1 -9138.745,E2 -9138.745} C_VEL
LIN {X 0,Y 439.372,Z 300.75,A -85,B 0,C 180,E1 -9141.609,E2 -9141.609} C_VEL
LIN {X 0,Y 439.402,Z 300.753,A -85,B 0,C 180,E1 -9144.844,E2 -9144.844} C_VEL
LIN {X 0,Y 439.376,Z 300.75,A -85,B 0,C 180,E1 -9148.14,E2 -9148.14} C_VEL
LIN {X 0,Y 439.413,Z 300.746,A -85,B 0,C 180,E1 -9151.604,E2 -9151.604} C_VEL
LIN {X 0,Y 439.381,Z 300.749,A -85,B 0,C 180,E1 -9154.413,E2 -9154.413} C_VEL
LIN {X 0,Y 439.367,Z 300.756,A -85,B 0,C 180,E1 -9157.424,E2 -9157.424} C_VEL
LIN {X 0,Y 439.445,Z 300.741,A -85,B 0,C 180,E1 -9160.663,E2 -9160.663} C_VEL
LIN {X 0,Y 439.466,Z 300.739,A -85,B 0,C 180,E1 -9164.224,E2 -9164.224} C_VEL
LIN {X 0,Y 439.487,Z 300.739,A -85,B 0,C 180,E1 -9168.001,E2 -9168.001} C_VEL
LIN {X 0,Y 439.506,Z 300.741,A -85,B 0,C 180,E1 -9171.725,E2 -9171.725} C_VEL
LIN {X 0,Y 439.616,Z 300.721,A -85,B 0,C 180,E1 -9174.495,E2 -9174.495} C_VEL
LIN {X 0,Y 439.634,Z 300.724,A -85,B 0,C 180,E1 -9178.168,E2 -9178.168} C_VEL
LIN {X 0,Y 439.762,Z 300.708,A -85,B 0,C 180,E1 -9180,E2 -9180} C_VEL
LIN {X 0,Y 439.634,Z 300.719,A -85,B 0,C 180,E1 -9182.749,E2 -9182.749} C_VEL
LIN {X 0,Y 439.567,Z 300.733,A -85,B 0,C 180,E1 -9186.426,E2 -9186.426} C_VEL
LIN {X 0,Y 439.499,Z 300.734,A -85,B 0,C 180,E1 -9189.201,E2 -9189.201} C_VEL
LIN {X 0,Y 439.469,Z 300.741,A -85,B 0,C 180,E1 -9192.937,E2 -9192.937} C_VEL
LIN {X 0,Y 439.45,Z 300.743,A -85,B 0,C 180,E1 -9196.348,E2 -9196.348} C_VEL
LIN {X 0,Y 439.405,Z 300.746,A -85,B 0,C 180,E1 -9199.626,E2 -9199.626} C_VEL
LIN {X 0,Y 439.366,Z 300.754,A -85,B 0,C 180,E1 -9202.575,E2 -9202.575} C_VEL
LIN {X 0,Y 439.382,Z 300.751,A -85,B 0,C 180,E1 -9205.586,E2 -9205.586} C_VEL
LIN {X 0,Y 439.402,Z 300.748,A -85,B 0,C 180,E1 -9208.674,E2 -9208.674} C_VEL
LIN {X 0,Y 439.371,Z 300.751,A -85,B 0,C 180,E1 -9212.03,E2 -9212.03} C_VEL
LIN {X 0,Y 439.393,Z 300.754,A -85,B 0,C 180,E1 -9215.339,E2 -9215.339} C_VEL
LIN {X 0,Y 439.371,Z 300.75,A -85,B 0,C 180,E1 -9218.596,E2 -9218.596} C_VEL
LIN {X 0,Y 439.383,Z 300.751,A -85,B 0,C 180,E1 -9221.255,E2 -9221.255} C_VEL
LIN {X 0,Y 439.4,Z 300.746,A -85,B 0,C 180,E1 -9224.729,E2 -9224.729} C_VEL
LIN {X 0,Y 439.386,Z 300.754,A -85,B 0,C 180,E1 -9227.794,E2 -9227.794} C_VEL
LIN {X 0,Y 439.39,Z 300.753,A -85,B 0,C 180,E1 -9230.223,E2 -9230.223} C_VEL
LIN {X 0,Y 439.373,Z 300.752,A -85,B 0,C 180,E1 -9233.712,E2 -9233.712} C_VEL
LIN {X 0,Y 439.374,Z 300.75,A -85,B 0,C 180,E1 -9237.053,E2 -9237.053} C_VEL
LIN {X 0,Y 439.379,Z 300.755,A -85,B 0,C 180,E1 -9240.273,E2 -9240.273} C_VEL
LIN {X 0,Y 439.383,Z 300.748,A -85,B 0,C 180,E1 -9243.393,E2 -9243.393} C_VEL
LIN {X 0,Y 439.383,Z 300.754,A -85,B 0,C 180,E1 -9246.429,E2 -9246.429} C_VEL
LIN {X 0,Y 439.389,Z 300.749,A -85,B 0,C 180,E1 -9249.396,E2 -9249.396} C_VEL
LIN {X 0,Y 439.405,Z 300.747,A -85,B 0,C 180,E1 -9252.308,E2 -9252.308} C_VEL
LIN {X 0,Y 439.447,Z 300.746,A -85,B 0,C 180,E1 -9255.173,E2 -9255.173} C_VEL
LIN {X 0,Y 439.483,Z 300.736,A -85,B 0,C 180,E1 -9258.001,E2 -9258.001} C_VEL
LIN {X 0,Y 439.504,Z 300.742,A -85,B 0,C 180,E1 -9261.725,E2 -9261.725} C_VEL
LIN {X 0,Y 439.574,Z 301.158,A -85,B 0,C 180,E1 -9261.897,E2 -9261.897} C_VEL
LIN {X 0,Y 440.783,Z 308.806,A -85,B 0,C 180,E1 -9263.591,E2 -9263.591} C_VEL
LIN {X 0,Y 440.528,Z 320.805,A -85,B 0,C 180,E1 -9266.111,E2 -9266.111} C_VEL
LIN {X 0,Y 443.916,Z 339.527,A -85,B 0,C 180,E1 -9266.552,E2 -9266.552} C_VEL
LIN {X 0,Y 443.887,Z 343.482,A -85,B 0,C 180,E1 -9266.617,E2 -9266.617} C_VEL
LIN {X 0,Y 443.209,Z 349.325,A -85,B 0,C 180,E1 -9266.69,E2 -9266.69} C_VEL
LIN {X 0,Y 437.472,Z 368.311,A -85,B 0,C 180,E1 -9266.801,E2 -9266.801} C_VEL
LIN {X 0,Y 436.76,Z 374.156,A -85,B 0,C 180,E1 -9266.875,E2 -9266.875} C_VEL
LIN {X 0,Y 436.119,Z 429.084,A -85,B 0,C 180,E1 -9267.805,E2 -9267.805} C_VEL
LIN {X 0,Y 435.787,Z 441.967,A -85,B 0,C 180,E1 -9268.209,E2 -9268.209} C_VEL
LIN {X 0,Y 435.364,Z 454.443,A -85,B 0,C 180,E1 -9268.785,E2 -9268.785} C_VEL
LIN {X 0,Y 434.791,Z 466.386,A -85,B 0,C 180,E1 -9269.536,E2 -9269.536} C_VEL
LIN {X 0,Y 434.152,Z 477.803,A -85,B 0,C 180,E1 -9270.463,E2 -9270.463} C_VEL
LIN {X 0,Y 433.488,Z 488.105,A -85,B 0,C 180,E1 -9271.509,E2 -9271.509} C_VEL
LIN {X 0,Y 432.973,Z 496.523,A -85,B 0,C 180,E1 -9272.558,E2 -9272.558} C_VEL
LIN {X 0,Y 432.381,Z 505.661,A -85,B 0,C 180,E1 -9273.96,E2 -9273.96} C_VEL
LIN {X 0,Y 431.899,Z 513.031,A -85,B 0,C 180,E1 -9275.368,E2 -9275.368} C_VEL
LIN {X 0,Y 431.702,Z 518.835,A -85,B 0,C 180,E1 -9276.754,E2 -9276.754} C_VEL
LIN {X 0,Y 431.417,Z 524.264,A -85,B 0,C 180,E1 -9278.43,E2 -9278.43} C_VEL
LIN {X 0,Y 431.326,Z 526.629,A -85,B 0,C 180,E1 -9279.377,E2 -9279.377} C_VEL
LIN {X 0,Y 431.248,Z 528.565,A -85,B 0,C 180,E1 -9280.326,E2 -9280.326} C_VEL
LIN {X 0,Y 431.174,Z 530.934,A -85,B 0,C 180,E1 -9282.047,E2 -9282.047} C_VEL
LIN {X 0,Y 431.088,Z 531.743,A -85,B 0,C 180,E1 -9283.193,E2 -9283.193} C_VEL
LIN {X 0,Y 431.069,Z 531.991,A -85,B 0,C 180,E1 -9284.155,E2 -9284.155} C_VEL
LIN {X 0,Y 431.154,Z 531.314,A -85,B 0,C 180,E1 -9285.904,E2 -9285.904} C_VEL
LIN {X 0,Y 431.15,Z 530.126,A -85,B 0,C 180,E1 -9287.061,E2 -9287.061} C_VEL
LIN {X 0,Y 431.256,Z 528.634,A -85,B 0,C 180,E1 -9288.036,E2 -9288.036} C_VEL
LIN {X 0,Y 431.457,Z 525.637,A -85,B 0,C 180,E1 -9289.457,E2 -9289.457} C_VEL
LIN {X 0,Y 431.681,Z 521.21,A -85,B 0,C 180,E1 -9290.987,E2 -9290.987} C_VEL
LIN {X 0,Y 432.06,Z 515.606,A -85,B 0,C 180,E1 -9292.472,E2 -9292.472} C_VEL
LIN {X 0,Y 432.579,Z 508.496,A -85,B 0,C 180,E1 -9293.963,E2 -9293.963} C_VEL
LIN {X 0,Y 433.065,Z 501.135,A -85,B 0,C 180,E1 -9295.213,E2 -9295.213} C_VEL
LIN {X 0,Y 433.723,Z 492.104,A -85,B 0,C 180,E1 -9296.461,E2 -9296.461} C_VEL
LIN {X 0,Y 434.413,Z 482.421,A -85,B 0,C 180,E1 -9297.547,E2 -9297.547} C_VEL
LIN {X 0,Y 435.074,Z 472.442,A -85,B 0,C 180,E1 -9298.458,E2 -9298.458} C_VEL
LIN {X 0,Y 435.791,Z 460.584,A -85,B 0,C 180,E1 -9299.319,E2 -9299.319} C_VEL
LIN {X 0,Y 436.298,Z 449.061,A -85,B 0,C 180,E1 -9299.956,E2 -9299.956} C_VEL
LIN {X 0,Y 436.738,Z 436.459,A -85,B 0,C 180,E1 -9300.456,E2 -9300.456} C_VEL
LIN {X 0,Y 437.018,Z 424.163,A -85,B 0,C 180,E1 -9300.769,E2 -9300.769} C_VEL
LIN {X 0,Y 437.99,Z 339.576,A -85,B 0,C 180,E1 -9302.186,E2 -9302.186} C_VEL
LIN {X 0,Y 434.056,Z 320.857,A -85,B 0,C 180,E1 -9302.725,E2 -9302.725} C_VEL
LIN {X 0,Y 434.344,Z 312.389,A -85,B 0,C 180,E1 -9304.493,E2 -9304.493} C_VEL
LIN {X 0,Y 433.161,Z 305.554,A -85,B 0,C 180,E1 -9306.024,E2 -9306.024} C_VEL
LIN {X 0,Y 432.294,Z 301.64,A -85,B 0,C 180,E1 -9306.978,E2 -9306.978} C_VEL
LIN {X 0,Y 432.284,Z 301.638,A -85,B 0,C 180,E1 -9310.172,E2 -9310.172} C_VEL
LIN {X 0,Y 432.307,Z 301.638,A -85,B 0,C 180,E1 -9313.061,E2 -9313.061} C_VEL
LIN {X 0,Y 432.325,Z 301.632,A -85,B 0,C 180,E1 -9315.664,E2 -9315.664} C_VEL
LIN {X 0,Y 432.303,Z 301.632,A -85,B 0,C 180,E1 -9318.401,E2 -9318.401} C_VEL
LIN {X 0,Y 432.324,Z 301.63,A -85,B 0,C 180,E1 -9321.849,E2 -9321.849} C_VEL
LIN {X 0,Y 432.32,Z 301.625,A -85,B 0,C 180,E1 -9325.321,E2 -9325.321} C_VEL
LIN {X 0,Y 432.31,Z 301.632,A -85,B 0,C 180,E1 -9328.653,E2 -9328.653} C_VEL
LIN {X 0,Y 432.333,Z 301.633,A -85,B 0,C 180,E1 -9331.874,E2 -9331.874} C_VEL
LIN {X 0,Y 432.312,Z 301.629,A -85,B 0,C 180,E1 -9334.997,E2 -9334.997} C_VEL
LIN {X 0,Y 432.348,Z 301.627,A -85,B 0,C 180,E1 -9338.045,E2 -9338.045} C_VEL
LIN {X 0,Y 432.372,Z 301.622,A -85,B 0,C 180,E1 -9341.029,E2 -9341.029} C_VEL
LIN {X 0,Y 432.378,Z 301.628,A -85,B 0,C 180,E1 -9343.959,E2 -9343.959} C_VEL
LIN {X 0,Y 432.444,Z 301.613,A -85,B 0,C 180,E1 -9347.803,E2 -9347.803} C_VEL
LIN {X 0,Y 432.435,Z 301.61,A -85,B 0,C 180,E1 -9351.589,E2 -9351.589} C_VEL
LIN {X 0,Y 432.535,Z 301.607,A -85,B 0,C 180,E1 -9354.406,E2 -9354.406} C_VEL
LIN {X 0,Y 432.583,Z 301.596,A -85,B 0,C 180,E1 -9358.138,E2 -9358.138} C_VEL
LIN {X 0,Y 432.535,Z 301.6,A -85,B 0,C 180,E1 -9360.931,E2 -9360.931} C_VEL
LIN {X 0,Y 432.544,Z 301.601,A -85,B 0,C 180,E1 -9362.794,E2 -9362.794} C_VEL
LIN {X 0,Y 432.573,Z 301.597,A -85,B 0,C 180,E1 -9365.594,E2 -9365.594} C_VEL
LIN {X 0,Y 432.44,Z 301.609,A -85,B 0,C 180,E1 -9368.411,E2 -9368.411} C_VEL
LIN {X 0,Y 432.449,Z 301.611,A -85,B 0,C 180,E1 -9372.197,E2 -9372.197} C_VEL
LIN {X 0,Y 432.42,Z 301.615,A -85,B 0,C 180,E1 -9376.04,E2 -9376.04} C_VEL
LIN {X 0,Y 432.378,Z 301.623,A -85,B 0,C 180,E1 -9379.485,E2 -9379.485} C_VEL
LIN {X 0,Y 432.303,Z 301.63,A -85,B 0,C 180,E1 -9382.965,E2 -9382.965} C_VEL
LIN {X 0,Y 432.312,Z 301.629,A -85,B 0,C 180,E1 -9386.036,E2 -9386.036} C_VEL
LIN {X 0,Y 432.324,Z 301.632,A -85,B 0,C 180,E1 -9389.189,E2 -9389.189} C_VEL
LIN {X 0,Y 432.316,Z 301.628,A -85,B 0,C 180,E1 -9392.444,E2 -9392.444} C_VEL
LIN {X 0,Y 432.337,Z 301.63,A -85,B 0,C 180,E1 -9395.632,E2 -9395.632} C_VEL
LIN {X 0,Y 432.319,Z 301.627,A -85,B 0,C 180,E1 -9398.713,E2 -9398.713} C_VEL
LIN {X 0,Y 432.315,Z 301.63,A -85,B 0,C 180,E1 -9401.8,E2 -9401.8} C_VEL
LIN {X 0,Y 432.329,Z 301.628,A -85,B 0,C 180,E1 -9404.348,E2 -9404.348} C_VEL
LIN {X 0,Y 432.312,Z 301.633,A -85,B 0,C 180,E1 -9407.017,E2 -9407.017} C_VEL
LIN {X 0,Y 432.328,Z 301.635,A -85,B 0,C 180,E1 -9409.822,E2 -9409.822} C_VEL
LIN {X 0,Y 432.301,Z 301.633,A -85,B 0,C 180,E1 -9413.023,E2 -9413.023} C_VEL
LIN {X 0,Y 432.357,Z 301.626,A -85,B 0,C 180,E1 -9415.998,E2 -9415.998} C_VEL
LIN {X 0,Y 432.345,Z 301.631,A -85,B 0,C 180,E1 -9419.491,E2 -9419.491} C_VEL
LIN {X 0,Y 432.418,Z 301.642,A -85,B 0,C 180,E1 -9422.899,E2 -9422.899} C_VEL
LIN {X 0,Y 434.951,Z 314.369,A -85,B 0,C 180,E1 -9425.669,E2 -9425.669} C_VEL
LIN {X 0,Y 435.341,Z 318.14,A -85,B 0,C 180,E1 -9426.449,E2 -9426.449} C_VEL
LIN {X 0,Y 434.122,Z 337.071,A -85,B 0,C 180,E1 -9430.126,E2 -9430.126} C_VEL
LIN {X 0,Y 433.761,Z 343.253,A -85,B 0,C 180,E1 -9431.312,E2 -9431.312} C_VEL
LIN {X 0,Y 437.276,Z 363.806,A -85,B 0,C 180,E1 -9431.855,E2 -9431.855} C_VEL
LIN {X 0,Y 437.75,Z 369.382,A -85,B 0,C 180,E1 -9431.974,E2 -9431.974} C_VEL
LIN {X 0,Y 436.9,Z 451.985,A -85,B 0,C 180,E1 -9433.381,E2 -9433.381} C_VEL
LIN {X 0,Y 436.352,Z 465.053,A -85,B 0,C 180,E1 -9433.78,E2 -9433.78} C_VEL
LIN {X 0,Y 435.728,Z 478.208,A -85,B 0,C 180,E1 -9434.387,E2 -9434.387} C_VEL
LIN {X 0,Y 435.025,Z 490.078,A -85,B 0,C 180,E1 -9435.14,E2 -9435.14} C_VEL
LIN {X 0,Y 434.189,Z 501.998,A -85,B 0,C 180,E1 -9436.117,E2 -9436.117} C_VEL
LIN {X 0,Y 433.593,Z 511.777,A -85,B 0,C 180,E1 -9437.123,E2 -9437.123} C_VEL
LIN {X 0,Y 432.945,Z 521.046,A -85,B 0,C 180,E1 -9438.294,E2 -9438.294} C_VEL
LIN {X 0,Y 432.304,Z 530.055,A -85,B 0,C 180,E1 -9439.699,E2 -9439.699} C_VEL
LIN {X 0,Y 431.836,Z 537.33,A -85,B 0,C 180,E1 -9441.107,E2 -9441.107} C_VEL
LIN {X 0,Y 431.535,Z 543.168,A -85,B 0,C 180,E1 -9442.515,E2 -9442.515} C_VEL
LIN {X 0,Y 431.287,Z 548.046,A -85,B 0,C 180,E1 -9444.019,E2 -9444.019} C_VEL
LIN {X 0,Y 431.27,Z 551.284,A -85,B 0,C 180,E1 -9445.327,E2 -9445.327} C_VEL
LIN {X 0,Y 431.186,Z 553.058,A -85,B 0,C 180,E1 -9446.263,E2 -9446.263} C_VEL
LIN {X 0,Y 431.235,Z 554.41,A -85,B 0,C 180,E1 -9447.198,E2 -9447.198} C_VEL
LIN {X 0,Y 431.203,Z 555.366,A -85,B 0,C 180,E1 -9448.133,E2 -9448.133} C_VEL
LIN {X 0,Y 431.169,Z 555.935,A -85,B 0,C 180,E1 -9449.067,E2 -9449.067} C_VEL
LIN {X 0,Y 431.168,Z 556.075,A -85,B 0,C 180,E1 -9450.001,E2 -9450.001} C_VEL
LIN {X 0,Y 431.203,Z 555.165,A -85,B 0,C 180,E1 -9451.869,E2 -9451.869} C_VEL
LIN {X 0,Y 431.237,Z 554.127,A -85,B 0,C 180,E1 -9452.803,E2 -9452.803} C_VEL
LIN {X 0,Y 431.188,Z 552.641,A -85,B 0,C 180,E1 -9453.739,E2 -9453.739} C_VEL
LIN {X 0,Y 431.295,Z 549.615,A -85,B 0,C 180,E1 -9455.143,E2 -9455.143} C_VEL
LIN {X 0,Y 431.377,Z 545.522,A -85,B 0,C 180,E1 -9456.549,E2 -9456.549} C_VEL
LIN {X 0,Y 431.616,Z 539.234,A -85,B 0,C 180,E1 -9458.192,E2 -9458.192} C_VEL
LIN {X 0,Y 431.958,Z 532.383,A -85,B 0,C 180,E1 -9459.601,E2 -9459.601} C_VEL
LIN {X 0,Y 432.434,Z 523.834,A -85,B 0,C 180,E1 -9461.01,E2 -9461.01} C_VEL
LIN {X 0,Y 433.016,Z 515.036,A -85,B 0,C 180,E1 -9462.181,E2 -9462.181} C_VEL
LIN {X 0,Y 433.664,Z 504.348,A -85,B 0,C 180,E1 -9463.338,E2 -9463.338} C_VEL
LIN {X 0,Y 434.298,Z 493.341,A -85,B 0,C 180,E1 -9464.288,E2 -9464.288} C_VEL
LIN {X 0,Y 434.91,Z 481.137,A -85,B 0,C 180,E1 -9465.105,E2 -9465.105} C_VEL
LIN {X 0,Y 435.449,Z 469.68,A -85,B 0,C 180,E1 -9465.685,E2 -9465.685} C_VEL
LIN {X 0,Y 435.915,Z 456.813,A -85,B 0,C 180,E1 -9466.148,E2 -9466.148} C_VEL
LIN {X 0,Y 436.166,Z 443.109,A -85,B 0,C 180,E1 -9466.439,E2 -9466.439} C_VEL
LIN {X 0,Y 436.811,Z 366.172,A -85,B 0,C 180,E1 -9467.709,E2 -9467.709} C_VEL
LIN {X 0,Y 433.379,Z 343.608,A -85,B 0,C 180,E1 -9468.221,E2 -9468.221} C_VEL
LIN {X 0,Y 434.334,Z 325.841,A -85,B 0,C 180,E1 -9471.6,E2 -9471.6} C_VEL
LIN {X 0,Y 434.859,Z 315.553,A -85,B 0,C 180,E1 -9473.579,E2 -9473.579} C_VEL
LIN {X 0,Y 433.038,Z 305.078,A -85,B 0,C 180,E1 -9475.731,E2 -9475.731} C_VEL
LIN {X 0,Y 432.394,Z 301.625,A -85,B 0,C 180,E1 -9476.465,E2 -9476.465} C_VEL
LIN {X 0,Y 432.347,Z 301.628,A -85,B 0,C 180,E1 -9479.188,E2 -9479.188} C_VEL
LIN {X 0,Y 432.327,Z 301.629,A -85,B 0,C 180,E1 -9482.443,E2 -9482.443} C_VEL
LIN {X 0,Y 432.348,Z 301.628,A -85,B 0,C 180,E1 -9485.632,E2 -9485.632} C_VEL
LIN {X 0,Y 432.329,Z 301.629,A -85,B 0,C 180,E1 -9488.712,E2 -9488.712} C_VEL
LIN {X 0,Y 432.324,Z 301.63,A -85,B 0,C 180,E1 -9491.799,E2 -9491.799} C_VEL
LIN {X 0,Y 432.338,Z 301.635,A -85,B 0,C 180,E1 -9494.348,E2 -9494.348} C_VEL
LIN {X 0,Y 432.321,Z 301.63,A -85,B 0,C 180,E1 -9497.016,E2 -9497.016} C_VEL
LIN {X 0,Y 432.336,Z 301.627,A -85,B 0,C 180,E1 -9499.821,E2 -9499.821} C_VEL
LIN {X 0,Y 432.309,Z 301.633,A -85,B 0,C 180,E1 -9503.022,E2 -9503.022} C_VEL
LIN {X 0,Y 432.363,Z 301.623,A -85,B 0,C 180,E1 -9505.997,E2 -9505.997} C_VEL
LIN {X 0,Y 432.35,Z 301.626,A -85,B 0,C 180,E1 -9509.49,E2 -9509.49} C_VEL
LIN {X 0,Y 432.351,Z 301.624,A -85,B 0,C 180,E1 -9511.874,E2 -9511.874} C_VEL
LIN {X 0,Y 432.381,Z 301.624,A -85,B 0,C 180,E1 -9515.539,E2 -9515.539} C_VEL
LIN {X 0,Y 432.355,Z 301.629,A -85,B 0,C 180,E1 -9519.046,E2 -9519.046} C_VEL
LIN {X 0,Y 432.365,Z 301.624,A -85,B 0,C 180,E1 -9522.01,E2 -9522.01} C_VEL
LIN {X 0,Y 432.398,Z 301.62,A -85,B 0,C 180,E1 -9524.926,E2 -9524.926} C_VEL
LIN {X 0,Y 432.463,Z 301.617,A -85,B 0,C 180,E1 -9527.803,E2 -9527.803} C_VEL
LIN {X 0,Y 432.466,Z 301.616,A -85,B 0,C 180,E1 -9531.59,E2 -9531.59} C_VEL
LIN {X 0,Y 432.592,Z 301.596,A -85,B 0,C 180,E1 -9534.406,E2 -9534.406} C_VEL
LIN {X 0,Y 432.603,Z 301.6,A -85,B 0,C 180,E1 -9538.138,E2 -9538.138} C_VEL
LIN {X 0,Y 432.731,Z 301.584,A -85,B 0,C 180,E1 -9540,E2 -9540} C_VEL
LIN {X 0,Y 432.585,Z 301.597,A -85,B 0,C 180,E1 -9542.793,E2 -9542.793} C_VEL
LIN {X 0,Y 432.581,Z 301.596,A -85,B 0,C 180,E1 -9545.594,E2 -9545.594} C_VEL
LIN {X 0,Y 432.467,Z 301.618,A -85,B 0,C 180,E1 -9548.41,E2 -9548.41} C_VEL
LIN {X 0,Y 432.462,Z 301.614,A -85,B 0,C 180,E1 -9552.196,E2 -9552.196} C_VEL
LIN {X 0,Y 432.434,Z 301.615,A -85,B 0,C 180,E1 -9556.039,E2 -9556.039} C_VEL
LIN {X 0,Y 432.39,Z 301.621,A -85,B 0,C 180,E1 -9559.485,E2 -9559.485} C_VEL
LIN {X 0,Y 432.32,Z 301.637,A -85,B 0,C 180,E1 -9562.964,E2 -9562.964} C_VEL
LIN {X 0,Y 432.342,Z 301.633,A -85,B 0,C 180,E1 -9565.002,E2 -9565.002} C_VEL
LIN {X 0,Y 432.349,Z 301.624,A -85,B 0,C 180,E1 -9568.125,E2 -9568.125} C_VEL
LIN {X 0,Y 432.323,Z 301.636,A -85,B 0,C 180,E1 -9571.346,E2 -9571.346} C_VEL
LIN {X 0,Y 432.339,Z 301.626,A -85,B 0,C 180,E1 -9574.677,E2 -9574.677} C_VEL
LIN {X 0,Y 432.334,Z 301.628,A -85,B 0,C 180,E1 -9578.15,E2 -9578.15} C_VEL
LIN {X 0,Y 432.326,Z 301.634,A -85,B 0,C 180,E1 -9581.6,E2 -9581.6} C_VEL
LIN {X 0,Y 432.335,Z 301.628,A -85,B 0,C 180,E1 -9584.347,E2 -9584.347} C_VEL
LIN {X 0,Y 432.318,Z 301.628,A -85,B 0,C 180,E1 -9587.016,E2 -9587.016} C_VEL
LIN {X 0,Y 432.315,Z 301.634,A -85,B 0,C 180,E1 -9589.823,E2 -9589.823} C_VEL
LIN {X 0,Y 432.306,Z 301.63,A -85,B 0,C 180,E1 -9593.021,E2 -9593.021} C_VEL
LIN {X 0,Y 432.361,Z 301.628,A -85,B 0,C 180,E1 -9595.996,E2 -9595.996} C_VEL
LIN {X 0,Y 432.348,Z 301.625,A -85,B 0,C 180,E1 -9599.489,E2 -9599.489} C_VEL
LIN {X 0,Y 432.349,Z 301.626,A -85,B 0,C 180,E1 -9601.874,E2 -9601.874} C_VEL
LIN {X 0,Y 432.378,Z 301.621,A -85,B 0,C 180,E1 -9605.538,E2 -9605.538} C_VEL
LIN {X 0,Y 432.351,Z 301.629,A -85,B 0,C 180,E1 -9609.045,E2 -9609.045} C_VEL
LIN {X 0,Y 432.361,Z 301.623,A -85,B 0,C 180,E1 -9612.01,E2 -9612.01} C_VEL
LIN {X 0,Y 432.395,Z 301.627,A -85,B 0,C 180,E1 -9614.926,E2 -9614.926} C_VEL
LIN {X 0,Y 432.459,Z 301.612,A -85,B 0,C 180,E1 -9617.803,E2 -9617.803} C_VEL
LIN {X 0,Y 432.468,Z 301.633,A -85,B 0,C 180,E1 -9621.634,E2 -9621.634} C_VEL
LIN {X 0,Y 433.818,Z 309.858,A -85,B 0,C 180,E1 -9623.488,E2 -9623.488} C_VEL
LIN {X 0,Y 433.588,Z 320.865,A -85,B 0,C 180,E1 -9625.831,E2 -9625.831} C_VEL
LIN {X 0,Y 437.069,Z 340.057,A -85,B 0,C 180,E1 -9626.311,E2 -9626.311} C_VEL
LIN {X 0,Y 436.76,Z 374.156,A -85,B 0,C 180,E1 -9626.875,E2 -9626.875} C_VEL
LIN {X 0,Y 436.063,Z 379.994,A -85,B 0,C 180,E1 -9626.948,E2 -9626.948} C_VEL
LIN {X 0,Y 430.354,Z 398.965,A -85,B 0,C 180,E1 -9627.068,E2 -9627.068} C_VEL
LIN {X 0,Y 429.599,Z 404.804,A -85,B 0,C 180,E1 -9627.141,E2 -9627.141} C_VEL
LIN {X 0,Y 429.237,Z 429.994,A -85,B 0,C 180,E1 -9627.596,E2 -9627.596} C_VEL
LIN {X 0,Y 428.856,Z 443.002,A -85,B 0,C 180,E1 -9628.019,E2 -9628.019} C_VEL
LIN {X 0,Y 428.44,Z 454.944,A -85,B 0,C 180,E1 -9628.589,E2 -9628.589} C_VEL
LIN {X 0,Y 427.894,Z 466.014,A -85,B 0,C 180,E1 -9629.293,E2 -9629.293} C_VEL
LIN {X 0,Y 427.206,Z 477.542,A -85,B 0,C 180,E1 -9630.235,E2 -9630.235} C_VEL
LIN {X 0,Y 426.555,Z 487.919,A -85,B 0,C 180,E1 -9631.297,E2 -9631.297} C_VEL
LIN {X 0,Y 425.993,Z 496.414,A -85,B 0,C 180,E1 -9632.363,E2 -9632.363} C_VEL
LIN {X 0,Y 425.463,Z 504.257,A -85,B 0,C 180,E1 -9633.551,E2 -9633.551} C_VEL
LIN {X 0,Y 424.957,Z 511.921,A -85,B 0,C 180,E1 -9634.98,E2 -9634.98} C_VEL
LIN {X 0,Y 424.666,Z 518.975,A -85,B 0,C 180,E1 -9636.652,E2 -9636.652} C_VEL
LIN {X 0,Y 424.389,Z 523.687,A -85,B 0,C 180,E1 -9638.091,E2 -9638.091} C_VEL
LIN {X 0,Y 424.21,Z 527.284,A -85,B 0,C 180,E1 -9639.535,E2 -9639.535} C_VEL
LIN {X 0,Y 424.141,Z 529.118,A -85,B 0,C 180,E1 -9640.501,E2 -9640.501} C_VEL
LIN {X 0,Y 424.088,Z 531.187,A -85,B 0,C 180,E1 -9642.11,E2 -9642.11} C_VEL
LIN {X 0,Y 423.98,Z 532.045,A -85,B 0,C 180,E1 -9643.418,E2 -9643.418} C_VEL
LIN {X 0,Y 423.972,Z 532.169,A -85,B 0,C 180,E1 -9644.397,E2 -9644.397} C_VEL
LIN {X 0,Y 424.058,Z 531.484,A -85,B 0,C 180,E1 -9646.004,E2 -9646.004} C_VEL
LIN {X 0,Y 424.084,Z 530.055,A -85,B 0,C 180,E1 -9647.354,E2 -9647.354} C_VEL
LIN {X 0,Y 424.216,Z 528.446,A -85,B 0,C 180,E1 -9648.346,E2 -9648.346} C_VEL
LIN {X 0,Y 424.419,Z 525.166,A -85,B 0,C 180,E1 -9649.843,E2 -9649.843} C_VEL
LIN {X 0,Y 424.691,Z 520.708,A -85,B 0,C 180,E1 -9651.349,E2 -9651.349} C_VEL
LIN {X 0,Y 425.113,Z 514.929,A -85,B 0,C 180,E1 -9652.86,E2 -9652.86} C_VEL
LIN {X 0,Y 425.688,Z 507.582,A -85,B 0,C 180,E1 -9654.376,E2 -9654.376} C_VEL
LIN {X 0,Y 426.249,Z 499.953,A -85,B 0,C 180,E1 -9655.645,E2 -9655.645} C_VEL
LIN {X 0,Y 426.92,Z 490.703,A -85,B 0,C 180,E1 -9656.901,E2 -9656.901} C_VEL
LIN {X 0,Y 427.716,Z 480.177,A -85,B 0,C 180,E1 -9658.056,E2 -9658.056} C_VEL
LIN {X 0,Y 428.45,Z 470.107,A -85,B 0,C 180,E1 -9658.939,E2 -9658.939} C_VEL
LIN {X 0,Y 429.119,Z 458.081,A -85,B 0,C 180,E1 -9659.771,E2 -9659.771} C_VEL
LIN {X 0,Y 429.7,Z 445.925,A -85,B 0,C 180,E1 -9660.404,E2 -9660.404} C_VEL
LIN {X 0,Y 430.132,Z 433.02,A -85,B 0,C 180,E1 -9660.873,E2 -9660.873} C_VEL
LIN {X 0,Y 430.457,Z 415.945,A -85,B 0,C 180,E1 -9661.222,E2 -9661.222} C_VEL
LIN {X 0,Y 431.333,Z 340.386,A -85,B 0,C 180,E1 -9662.507,E2 -9662.507} C_VEL
LIN {X 0,Y 427.213,Z 321.088,A -85,B 0,C 180,E1 -9663.076,E2 -9663.076} C_VEL
LIN {X 0,Y 427.366,Z 312.867,A -85,B 0,C 180,E1 -9664.828,E2 -9664.828} C_VEL
LIN {X 0,Y 425.293,Z 302.511,A -85,B 0,C 180,E1 -9667.244,E2 -9667.244} C_VEL
LIN {X 0,Y 425.24,Z 302.518,A -85,B 0,C 180,E1 -9670.514,E2 -9670.514} C_VEL
LIN {X 0,Y 425.248,Z 302.516,A -85,B 0,C 180,E1 -9673.35,E2 -9673.35} C_VEL
LIN {X 0,Y 425.251,Z 302.512,A -85,B 0,C 180,E1 -9676.043,E2 -9676.043} C_VEL
LIN {X 0,Y 425.246,Z 302.515,A -85,B 0,C 180,E1 -9679.483,E2 -9679.483} C_VEL
LIN {X 0,Y 425.268,Z 302.508,A -85,B 0,C 180,E1 -9682.488,E2 -9682.488} C_VEL
LIN {X 0,Y 425.278,Z 302.496,A -85,B 0,C 180,E1 -9685.815,E2 -9685.815} C_VEL
LIN {X 0,Y 425.282,Z 302.512,A -85,B 0,C 180,E1 -9689.239,E2 -9689.239} C_VEL
LIN {X 0,Y 425.259,Z 302.51,A -85,B 0,C 180,E1 -9692.436,E2 -9692.436} C_VEL
LIN {X 0,Y 425.31,Z 302.507,A -85,B 0,C 180,E1 -9695.6,E2 -9695.6} C_VEL
LIN {X 0,Y 425.283,Z 302.504,A -85,B 0,C 180,E1 -9698.681,E2 -9698.681} C_VEL
LIN {X 0,Y 425.303,Z 302.504,A -85,B 0,C 180,E1 -9701.702,E2 -9701.702} C_VEL
LIN {X 0,Y 425.29,Z 302.505,A -85,B 0,C 180,E1 -9704.669,E2 -9704.669} C_VEL
LIN {X 0,Y 425.399,Z 302.488,A -85,B 0,C 180,E1 -9707.598,E2 -9707.598} C_VEL
LIN {X 0,Y 425.384,Z 302.487,A -85,B 0,C 180,E1 -9711.449,E2 -9711.449} C_VEL
LIN {X 0,Y 425.493,Z 302.485,A -85,B 0,C 180,E1 -9714.313,E2 -9714.313} C_VEL
LIN {X 0,Y 425.552,Z 302.471,A -85,B 0,C 180,E1 -9718.107,E2 -9718.107} C_VEL
LIN {X 0,Y 425.498,Z 302.477,A -85,B 0,C 180,E1 -9720.947,E2 -9720.947} C_VEL
LIN {X 0,Y 425.5,Z 302.478,A -85,B 0,C 180,E1 -9722.84,E2 -9722.84} C_VEL
LIN {X 0,Y 425.529,Z 302.475,A -85,B 0,C 180,E1 -9725.687,E2 -9725.687} C_VEL
LIN {X 0,Y 425.388,Z 302.489,A -85,B 0,C 180,E1 -9728.551,E2 -9728.551} C_VEL
LIN {X 0,Y 425.403,Z 302.49,A -85,B 0,C 180,E1 -9732.402,E2 -9732.402} C_VEL
LIN {X 0,Y 425.379,Z 302.493,A -85,B 0,C 180,E1 -9736.312,E2 -9736.312} C_VEL
LIN {X 0,Y 425.32,Z 302.501,A -85,B 0,C 180,E1 -9739.636,E2 -9739.636} C_VEL
LIN {X 0,Y 425.279,Z 302.503,A -85,B 0,C 180,E1 -9742.339,E2 -9742.339} C_VEL
LIN {X 0,Y 425.253,Z 302.514,A -85,B 0,C 180,E1 -9745.448,E2 -9745.448} C_VEL
LIN {X 0,Y 425.305,Z 302.503,A -85,B 0,C 180,E1 -9748.862,E2 -9748.862} C_VEL
LIN {X 0,Y 425.258,Z 302.509,A -85,B 0,C 180,E1 -9751.928,E2 -9751.928} C_VEL
LIN {X 0,Y 425.292,Z 302.507,A -85,B 0,C 180,E1 -9755.337,E2 -9755.337} C_VEL
LIN {X 0,Y 425.274,Z 302.506,A -85,B 0,C 180,E1 -9758.902,E2 -9758.902} C_VEL
LIN {X 0,Y 425.274,Z 302.505,A -85,B 0,C 180,E1 -9761.957,E2 -9761.957} C_VEL
LIN {X 0,Y 425.28,Z 302.508,A -85,B 0,C 180,E1 -9765.284,E2 -9765.284} C_VEL
LIN {X 0,Y 425.263,Z 302.513,A -85,B 0,C 180,E1 -9768.622,E2 -9768.622} C_VEL
LIN {X 0,Y 425.288,Z 302.509,A -85,B 0,C 180,E1 -9771.102,E2 -9771.102} C_VEL
LIN {X 0,Y 425.296,Z 302.505,A -85,B 0,C 180,E1 -9774.665,E2 -9774.665} C_VEL
LIN {X 0,Y 425.262,Z 302.511,A -85,B 0,C 180,E1 -9778.074,E2 -9778.074} C_VEL
LIN {X 0,Y 425.329,Z 302.505,A -85,B 0,C 180,E1 -9781.369,E2 -9781.369} C_VEL
LIN {X 0,Y 425.387,Z 302.527,A -85,B 0,C 180,E1 -9782.586,E2 -9782.586} C_VEL
LIN {X 0,Y 427.799,Z 314.456,A -85,B 0,C 180,E1 -9785.242,E2 -9785.242} C_VEL
LIN {X 0,Y 428.454,Z 319.446,A -85,B 0,C 180,E1 -9786.306,E2 -9786.306} C_VEL
LIN {X 0,Y 427.242,Z 337.101,A -85,B 0,C 180,E1 -9789.792,E2 -9789.792} C_VEL
LIN {X 0,Y 426.884,Z 343.159,A -85,B 0,C 180,E1 -9790.968,E2 -9790.968} C_VEL
LIN {X 0,Y 430.571,Z 364.166,A -85,B 0,C 180,E1 -9791.531,E2 -9791.531} C_VEL
LIN {X 0,Y 431.105,Z 370.437,A -85,B 0,C 180,E1 -9791.668,E2 -9791.668} C_VEL
LIN {X 0,Y 430.187,Z 452.084,A -85,B 0,C 180,E1 -9793.083,E2 -9793.083} C_VEL
LIN {X 0,Y 429.662,Z 464.293,A -85,B 0,C 180,E1 -9793.459,E2 -9793.459} C_VEL
LIN {X 0,Y 429.005,Z 477.603,A -85,B 0,C 180,E1 -9794.075,E2 -9794.075} C_VEL
LIN {X 0,Y 428.276,Z 488.798,A -85,B 0,C 180,E1 -9794.779,E2 -9794.779} C_VEL
LIN {X 0,Y 427.443,Z 500.399,A -85,B 0,C 180,E1 -9795.723,E2 -9795.723} C_VEL
LIN {X 0,Y 426.743,Z 510.847,A -85,B 0,C 180,E1 -9796.792,E2 -9796.792} C_VEL
LIN {X 0,Y 426.146,Z 519.403,A -85,B 0,C 180,E1 -9797.863,E2 -9797.863} C_VEL
LIN {X 0,Y 425.449,Z 527.308,A -85,B 0,C 180,E1 -9799.05,E2 -9799.05} C_VEL
LIN {X 0,Y 424.949,Z 535.056,A -85,B 0,C 180,E1 -9800.481,E2 -9800.481} C_VEL
LIN {X 0,Y 424.541,Z 541.279,A -85,B 0,C 180,E1 -9801.912,E2 -9801.912} C_VEL
LIN {X 0,Y 424.306,Z 546.24,A -85,B 0,C 180,E1 -9803.343,E2 -9803.343} C_VEL
LIN {X 0,Y 424.207,Z 550.081,A -85,B 0,C 180,E1 -9804.773,E2 -9804.773} C_VEL
LIN {X 0,Y 424.098,Z 552.906,A -85,B 0,C 180,E1 -9806.2,E2 -9806.2} C_VEL
LIN {X 0,Y 424.13,Z 554.247,A -85,B 0,C 180,E1 -9807.151,E2 -9807.151} C_VEL
LIN {X 0,Y 424.129,Z 555.194,A -85,B 0,C 180,E1 -9808.102,E2 -9808.102} C_VEL
LIN {X 0,Y 424.088,Z 555.749,A -85,B 0,C 180,E1 -9809.051,E2 -9809.051} C_VEL
LIN {X 0,Y 424.085,Z 555.871,A -85,B 0,C 180,E1 -9810.001,E2 -9810.001} C_VEL
LIN {X 0,Y 424.129,Z 554.941,A -85,B 0,C 180,E1 -9811.9,E2 -9811.9} C_VEL
LIN {X 0,Y 424.133,Z 553.889,A -85,B 0,C 180,E1 -9812.85,E2 -9812.85} C_VEL
LIN {X 0,Y 424.099,Z 552.384,A -85,B 0,C 180,E1 -9813.802,E2 -9813.802} C_VEL
LIN {X 0,Y 424.207,Z 549.334,A -85,B 0,C 180,E1 -9815.229,E2 -9815.229} C_VEL
LIN {X 0,Y 424.301,Z 545.216,A -85,B 0,C 180,E1 -9816.659,E2 -9816.659} C_VEL
LIN {X 0,Y 424.547,Z 538.9,A -85,B 0,C 180,E1 -9818.329,E2 -9818.329} C_VEL
LIN {X 0,Y 424.926,Z 532.013,A -85,B 0,C 180,E1 -9819.761,E2 -9819.761} C_VEL
LIN {X 0,Y 425.318,Z 524.975,A -85,B 0,C 180,E1 -9820.955,E2 -9820.955} C_VEL
LIN {X 0,Y 425.924,Z 516.497,A -85,B 0,C 180,E1 -9822.146,E2 -9822.146} C_VEL
LIN {X 0,Y 426.601,Z 506.005,A -85,B 0,C 180,E1 -9823.336,E2 -9823.336} C_VEL
LIN {X 0,Y 427.196,Z 495.609,A -85,B 0,C 180,E1 -9824.287,E2 -9824.287} C_VEL
LIN {X 0,Y 427.852,Z 484.217,A -85,B 0,C 180,E1 -9825.116,E2 -9825.116} C_VEL
LIN {X 0,Y 428.429,Z 472.555,A -85,B 0,C 180,E1 -9825.766,E2 -9825.766} C_VEL
LIN {X 0,Y 428.941,Z 460.035,A -85,B 0,C 180,E1 -9826.265,E2 -9826.265} C_VEL
LIN {X 0,Y 429.261,Z 447.414,A -85,B 0,C 180,E1 -9826.589,E2 -9826.589} C_VEL
LIN {X 0,Y 429.994,Z 367.031,A -85,B 0,C 180,E1 -9827.941,E2 -9827.941} C_VEL
LIN {X 0,Y 426.429,Z 343.358,A -85,B 0,C 180,E1 -9828.498,E2 -9828.498} C_VEL
LIN {X 0,Y 427.528,Z 324.128,A -85,B 0,C 180,E1 -9832.216,E2 -9832.216} C_VEL
LIN {X 0,Y 427.888,Z 316.398,A -85,B 0,C 180,E1 -9833.73,E2 -9833.73} C_VEL
LIN {X 0,Y 425.361,Z 302.501,A -85,B 0,C 180,E1 -9836.685,E2 -9836.685} C_VEL
LIN {X 0,Y 425.295,Z 302.511,A -85,B 0,C 180,E1 -9839.72,E2 -9839.72} C_VEL
LIN {X 0,Y 425.287,Z 302.504,A -85,B 0,C 180,E1 -9843.048,E2 -9843.048} C_VEL
LIN {X 0,Y 425.286,Z 302.511,A -85,B 0,C 180,E1 -9845.929,E2 -9845.929} C_VEL
LIN {X 0,Y 425.266,Z 302.507,A -85,B 0,C 180,E1 -9849.038,E2 -9849.038} C_VEL
LIN {X 0,Y 425.273,Z 302.51,A -85,B 0,C 180,E1 -9852.654,E2 -9852.654} C_VEL
LIN {X 0,Y 425.265,Z 302.51,A -85,B 0,C 180,E1 -9856.044,E2 -9856.044} C_VEL
LIN {X 0,Y 425.28,Z 302.505,A -85,B 0,C 180,E1 -9859.481,E2 -9859.481} C_VEL
LIN {X 0,Y 425.28,Z 302.511,A -85,B 0,C 180,E1 -9862.489,E2 -9862.489} C_VEL
LIN {X 0,Y 425.311,Z 302.501,A -85,B 0,C 180,E1 -9865.817,E2 -9865.817} C_VEL
LIN {X 0,Y 425.294,Z 302.507,A -85,B 0,C 180,E1 -9869.239,E2 -9869.239} C_VEL
LIN {X 0,Y 425.304,Z 302.503,A -85,B 0,C 180,E1 -9872.439,E2 -9872.439} C_VEL
LIN {X 0,Y 425.349,Z 302.499,A -85,B 0,C 180,E1 -9875.602,E2 -9875.602} C_VEL
LIN {X 0,Y 425.297,Z 302.504,A -85,B 0,C 180,E1 -9878.681,E2 -9878.681} C_VEL
LIN {X 0,Y 425.326,Z 302.504,A -85,B 0,C 180,E1 -9881.702,E2 -9881.702} C_VEL
LIN {X 0,Y 425.351,Z 302.496,A -85,B 0,C 180,E1 -9884.671,E2 -9884.671} C_VEL
LIN {X 0,Y 425.416,Z 302.496,A -85,B 0,C 180,E1 -9887.598,E2 -9887.598} C_VEL
LIN {X 0,Y 425.411,Z 302.493,A -85,B 0,C 180,E1 -9891.449,E2 -9891.449} C_VEL
LIN {X 0,Y 425.547,Z 302.475,A -85,B 0,C 180,E1 -9894.313,E2 -9894.313} C_VEL
LIN {X 0,Y 425.573,Z 302.476,A -85,B 0,C 180,E1 -9898.107,E2 -9898.107} C_VEL
LIN {X 0,Y 425.7,Z 302.46,A -85,B 0,C 180,E1 -9900,E2 -9900} C_VEL
LIN {X 0,Y 425.539,Z 302.474,A -85,B 0,C 180,E1 -9902.84,E2 -9902.84} C_VEL
LIN {X 0,Y 425.483,Z 302.483,A -85,B 0,C 180,E1 -9906.549,E2 -9906.549} C_VEL
LIN {X 0,Y 425.401,Z 302.49,A -85,B 0,C 180,E1 -9909.509,E2 -9909.509} C_VEL
LIN {X 0,Y 425.397,Z 302.495,A -85,B 0,C 180,E1 -9912.903,E2 -9912.903} C_VEL
LIN {X 0,Y 425.364,Z 302.501,A -85,B 0,C 180,E1 -9916.604,E2 -9916.604} C_VEL
LIN {X 0,Y 425.331,Z 302.499,A -85,B 0,C 180,E1 -9919.635,E2 -9919.635} C_VEL
LIN {X 0,Y 425.291,Z 302.505,A -85,B 0,C 180,E1 -9922.338,E2 -9922.338} C_VEL
LIN {X 0,Y 425.323,Z 302.503,A -85,B 0,C 180,E1 -9924.657,E2 -9924.657} C_VEL
LIN {X 0,Y 425.302,Z 302.506,A -85,B 0,C 180,E1 -9927.561,E2 -9927.561} C_VEL
LIN {X 0,Y 425.29,Z 302.506,A -85,B 0,C 180,E1 -9930.816,E2 -9930.816} C_VEL
LIN {X 0,Y 425.311,Z 302.501,A -85,B 0,C 180,E1 -9934.287,E2 -9934.287} C_VEL
LIN {X 0,Y 425.279,Z 302.512,A -85,B 0,C 180,E1 -9937.694,E2 -9937.694} C_VEL
LIN {X 0,Y 425.278,Z 302.506,A -85,B 0,C 180,E1 -9940.519,E2 -9940.519} C_VEL
LIN {X 0,Y 425.263,Z 302.513,A -85,B 0,C 180,E1 -9943.955,E2 -9943.955} C_VEL
LIN {X 0,Y 425.272,Z 302.508,A -85,B 0,C 180,E1 -9947.346,E2 -9947.346} C_VEL
LIN {X 0,Y 425.274,Z 302.506,A -85,B 0,C 180,E1 -9950.96,E2 -9950.96} C_VEL
LIN {X 0,Y 425.283,Z 302.512,A -85,B 0,C 180,E1 -9954.071,E2 -9954.071} C_VEL
LIN {X 0,Y 425.284,Z 302.506,A -85,B 0,C 180,E1 -9956.951,E2 -9956.951} C_VEL
LIN {X 0,Y 425.288,Z 302.511,A -85,B 0,C 180,E1 -9960.279,E2 -9960.279} C_VEL
LIN {X 0,Y 425.302,Z 302.502,A -85,B 0,C 180,E1 -9963.501,E2 -9963.501} C_VEL
LIN {X 0,Y 425.305,Z 302.51,A -85,B 0,C 180,E1 -9966.634,E2 -9966.634} C_VEL
LIN {X 0,Y 425.329,Z 302.502,A -85,B 0,C 180,E1 -9970.364,E2 -9970.364} C_VEL
LIN {X 0,Y 425.389,Z 302.492,A -85,B 0,C 180,E1 -9973.688,E2 -9973.688} C_VEL
LIN {X 0,Y 425.412,Z 302.491,A -85,B 0,C 180,E1 -9977.597,E2 -9977.597} C_VEL
LIN {X 0,Y 425.438,Z 302.577,A -85,B 0,C 180,E1 -9981.473,E2 -9981.473} C_VEL
LIN {X 0,Y 426.847,Z 310.927,A -85,B 0,C 180,E1 -9983.381,E2 -9983.381} C_VEL
LIN {X 0,Y 426.617,Z 321.17,A -85,B 0,C 180,E1 -9985.591,E2 -9985.591} C_VEL
LIN {X 0,Y 430.239,Z 341.421,A -85,B 0,C 180,E1 -9986.08,E2 -9986.08} C_VEL
LIN {X 0,Y 429.599,Z 404.804,A -85,B 0,C 180,E1 -9987.141,E2 -9987.141} C_VEL
LIN {X 0,Y 428.834,Z 410.652,A -85,B 0,C 180,E1 -9987.209,E2 -9987.209} C_VEL
LIN {X 0,Y 422.963,Z 429.567,A -85,B 0,C 180,E1 -9987.361,E2 -9987.361} C_VEL
LIN {X 0,Y 422.171,Z 435.313,A -85,B 0,C 180,E1 -9987.505,E2 -9987.505} C_VEL
LIN {X 0,Y 421.783,Z 448.479,A -85,B 0,C 180,E1 -9988.025,E2 -9988.025} C_VEL
LIN {X 0,Y 421.29,Z 460.365,A -85,B 0,C 180,E1 -9988.685,E2 -9988.685} C_VEL
LIN {X 0,Y 420.649,Z 471.795,A -85,B 0,C 180,E1 -9989.52,E2 -9989.52} C_VEL
LIN {X 0,Y 419.908,Z 483.364,A -85,B 0,C 180,E1 -9990.598,E2 -9990.598} C_VEL
LIN {X 0,Y 419.269,Z 492.699,A -85,B 0,C 180,E1 -9991.68,E2 -9991.68} C_VEL
LIN {X 0,Y 418.637,Z 501.224,A -85,B 0,C 180,E1 -9992.886,E2 -9992.886} C_VEL
LIN {X 0,Y 418.106,Z 509.506,A -85,B 0,C 180,E1 -9994.337,E2 -9994.337} C_VEL
LIN {X 0,Y 417.726,Z 516.189,A -85,B 0,C 180,E1 -9995.793,E2 -9995.793} C_VEL
LIN {X 0,Y 417.465,Z 521.528,A -85,B 0,C 180,E1 -9997.253,E2 -9997.253} C_VEL
LIN {X 0,Y 417.214,Z 525.704,A -85,B 0,C 180,E1 -9998.719,E2 -9998.719} C_VEL
LIN {X 0,Y 417.095,Z 527.905,A -85,B 0,C 180,E1 -9999.7,E2 -9999.7} C_VEL
LIN {X 0,Y 417.048,Z 529.618,A -85,B 0,C 180,E1 -10000.682,E2 -10000.682} C_VEL
LIN {X 0,Y 416.999,Z 531.433,A -85,B 0,C 180,E1 -10002.173,E2 -10002.173} C_VEL
LIN {X 0,Y 416.884,Z 532.293,A -85,B 0,C 180,E1 -10003.651,E2 -10003.651} C_VEL
LIN {X 0,Y 416.895,Z 532.336,A -85,B 0,C 180,E1 -10004.646,E2 -10004.646} C_VEL
LIN {X 0,Y 416.969,Z 531.656,A -85,B 0,C 180,E1 -10006.11,E2 -10006.11} C_VEL
LIN {X 0,Y 417.033,Z 529.946,A -85,B 0,C 180,E1 -10007.657,E2 -10007.657} C_VEL
LIN {X 0,Y 417.301,Z 526.711,A -85,B 0,C 180,E1 -10009.417,E2 -10009.417} C_VEL
LIN {X 0,Y 417.6,Z 521.896,A -85,B 0,C 180,E1 -10011.212,E2 -10011.212} C_VEL
LIN {X 0,Y 418.026,Z 516.368,A -85,B 0,C 180,E1 -10012.747,E2 -10012.747} C_VEL
LIN {X 0,Y 418.585,Z 509.338,A -85,B 0,C 180,E1 -10014.289,E2 -10014.289} C_VEL
LIN {X 0,Y 419.175,Z 501.89,A -85,B 0,C 180,E1 -10015.607,E2 -10015.607} C_VEL
LIN {X 0,Y 419.884,Z 493.212,A -85,B 0,C 180,E1 -10016.866,E2 -10016.866} C_VEL
LIN {X 0,Y 420.689,Z 483.328,A -85,B 0,C 180,E1 -10018.024,E2 -10018.024} C_VEL
LIN {X 0,Y 421.539,Z 472.43,A -85,B 0,C 180,E1 -10019.049,E2 -10019.049} C_VEL
LIN {X 0,Y 422.212,Z 462.199,A -85,B 0,C 180,E1 -10019.82,E2 -10019.82} C_VEL
LIN {X 0,Y 422.843,Z 450.015,A -85,B 0,C 180,E1 -10020.533,E2 -10020.533} C_VEL
LIN {X 0,Y 423.362,Z 436.87,A -85,B 0,C 180,E1 -10021.074,E2 -10021.074} C_VEL
LIN {X 0,Y 423.661,Z 424.589,A -85,B 0,C 180,E1 -10021.397,E2 -10021.397} C_VEL
LIN {X 0,Y 424.819,Z 342.171,A -85,B 0,C 180,E1 -10022.818,E2 -10022.818} C_VEL
LIN {X 0,Y 421.284,Z 325.216,A -85,B 0,C 180,E1 -10023.318,E2 -10023.318} C_VEL
LIN {X 0,Y 420.368,Z 321.219,A -85,B 0,C 180,E1 -10023.461,E2 -10023.461} C_VEL
LIN {X 0,Y 420.452,Z 314.1,A -85,B 0,C 180,E1 -10025.01,E2 -10025.01} C_VEL
LIN {X 0,Y 418.237,Z 303.39,A -85,B 0,C 180,E1 -10027.568,E2 -10027.568} C_VEL
LIN {X 0,Y 418.203,Z 303.393,A -85,B 0,C 180,E1 -10030.949,E2 -10030.949} C_VEL
LIN {X 0,Y 418.201,Z 303.392,A -85,B 0,C 180,E1 -10033.728,E2 -10033.728} C_VEL
LIN {X 0,Y 418.195,Z 303.392,A -85,B 0,C 180,E1 -10036.447,E2 -10036.447} C_VEL
